KUKA KRL program: MyProgram_070().src

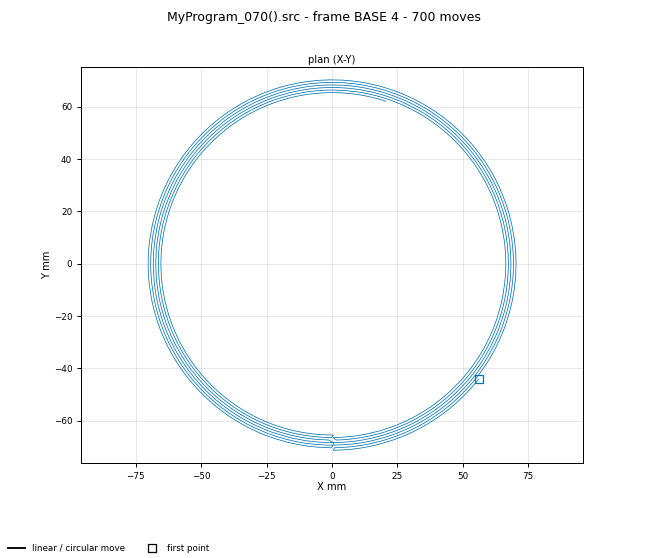
[picture p0: tool path of MyProgram_070().src in frame BASE 4, 700 of 700 moves have a stored position in this frame; points joined in program order, loops and branches not executed]
&ACCESS RVP
&REL 1
&PARAM TEMPLATE = C:\KRC\Roboter\Template\vorgabe
&PARAM EDITMASK = *
DEF MyProgram_070()
; ---- Setting reference (Base) ----
$BASE = BASE_DATA[4]

; --------------------------
; ---- Setting tool (TCP) ----
$TOOL = TOOL_DATA[3]
; --------------------------

$VEL.CP = VEL_APROX_PRINT
Startdeposition()
$VEL.CP = VEL_PRINT
LIN {X 56.046,Y -44.0463,Z 76,A -44.288,B 24.9035,C -2.2676,E1 25.1245,E2 128.6821} C_DIS
LIN {X 53.7927,Y -46.7714,Z 76,A -47.1061,B 24.9041,C -2.261,E1 25.1194,E2 131.503} C_DIS
LIN {X 51.1521,Y -49.6455,Z 76,A -50.0021,B 24.9041,C -2.2599,E1 25.1139,E2 134.3889} C_DIS
LIN {X 49.3417,Y -51.445,Z 76,A -52.3384,B 24.9053,C -2.2472,E1 25.1092,E2 136.7455} C_DIS
LIN {X 46.445,Y -54.0753,Z 76,A -55.3463,B 24.9056,C -2.2438,E1 25.1029,E2 139.7495} C_DIS
LIN {X 43.668,Y -56.3411,Z 76,A -58.1698,B 24.9059,C -2.2391,E1 25.0967,E2 142.5734} C_DIS
LIN {X 40.701,Y -58.5203,Z 76,A -60.9127,B 24.9059,C -2.239,E1 25.0905,E2 145.307} C_DIS
LIN {X 38.2526,Y -60.15,Z 76,A -63.889,B 24.9077,C -2.2179,E1 25.0835,E2 148.3235} C_DIS
LIN {X 34.8025,Y -62.2092,Z 76,A -67.0175,B 24.908,C -2.2149,E1 25.0759,E2 151.4498} C_DIS
LIN {X 30.8316,Y -64.2698,Z 76,A -70.4455,B 24.908,C -2.2135,E1 25.0673,E2 154.8717} C_DIS
LIN {X 27.6575,Y -65.6982,Z 76,A -73.0295,B 24.908,C -2.2151,E1 25.0607,E2 157.4458} C_DIS
LIN {X 23.6668,Y -67.239,Z 76,A -76.1249,B 24.9076,C -2.2196,E1 25.0527,E2 160.5239} C_DIS
LIN {X 19.5102,Y -68.5606,Z 76,A -79.8203,B 24.9083,C -2.2105,E1 25.0428,E2 164.2341} C_DIS
LIN {X 15.9897,Y -69.466,Z 76,A -83.1017,B 24.9094,C -2.1982,E1 25.0338,E2 167.5398} C_DIS
LIN {X 11.549,Y -70.341,Z 76,A -86.5042,B 24.9091,C -2.2014,E1 25.0245,E2 170.9309} C_DIS
LIN {X 7.3989,Y -70.8975,Z 76,A -90.297,B 24.9102,C -2.1885,E1 25.0139,E2 174.7517} C_DIS
LIN {X 3.8952,Y -71.176,Z 76,A -93.5754,B 24.9112,C -2.1759,E1 25.0047,E2 178.0587} C_DIS
LIN {X 0.4617,Y -71.2706,Z 76,A -93.732,B 24.9057,C -2.2418,E1 25.0047,E2 178.0587} C_DIS
Enddeposition()
LIN {X 0.4617,Y -71.2706,Z 76,A -93.732,B 24.9057,C -2.2418,E1 25.0047,E2 178.0587} C_DIS
Startdeposition()
$VEL.CP = VEL_PRINT
LIN {X 0.982,Y -70.3014,Z 76,A -93.6346,B 24.905,C -2.2498,E1 25.0051,E2 177.9423} C_DIS
LIN {X 4.084,Y -70.1891,Z 76,A -91.6184,B 24.9061,C -2.2376,E1 25.0106,E2 175.9557} C_DIS
LIN {X 7.1431,Y -69.944,Z 76,A -88.5948,B 24.9048,C -2.2524,E1 25.0191,E2 172.8989} C_DIS
LIN {X 11.0153,Y -69.4399,Z 76,A -85.5875,B 24.905,C -2.25,E1 25.0274,E2 169.8999} C_DIS
LIN {X 14.077,Y -68.8839,Z 76,A -83.2844,B 24.9054,C -2.246,E1 25.0337,E2 167.6089} C_DIS
LIN {X 18.31,Y -67.8815,Z 76,A -79.8324,B 24.9053,C -2.247,E1 25.043,E2 164.1596} C_DIS
LIN {X 22.0646,Y -66.756,Z 76,A -76.4652,B 24.9046,C -2.2553,E1 25.052,E2 160.7789} C_DIS
LIN {X 26.987,Y -64.9227,Z 76,A -72.2326,B 24.9042,C -2.2597,E1 25.0631,E2 156.545} C_DIS
LIN {X 30.316,Y -63.4359,Z 76,A -69.0283,B 24.9033,C -2.2706,E1 25.0712,E2 153.3231} C_DIS
LIN {X 33.2683,Y -61.9384,Z 76,A -66.4121,B 24.9031,C -2.2729,E1 25.0777,E2 150.7087} C_DIS
LIN {X 35.6896,Y -60.5757,Z 76,A -64.0683,B 24.9025,C -2.2791,E1 25.0834,E2 148.3573} C_DIS
LIN {X 39.2963,Y -58.3008,Z 76,A -61.2698,B 24.9036,C -2.2674,E1 25.0899,E2 145.5958} C_DIS
LIN {X 41.6342,Y -56.6548,Z 76,A -58.6689,B 24.9025,C -2.2794,E1 25.0958,E2 142.9754} C_DIS
LIN {X 43.4611,Y -55.2659,Z 76,A -56.6561,B 24.9018,C -2.2873,E1 25.1003,E2 140.9513} C_DIS
LIN {X 45.7398,Y -53.3953,Z 76,A -54.201,B 24.9013,C -2.2941,E1 25.1056,E2 138.4896} C_DIS
LIN {X 48.1424,Y -51.2392,Z 76,A -51.4487,B 24.9004,C -2.3035,E1 25.1112,E2 135.7262} C_DIS
LIN {X 50.9425,Y -48.4564,Z 76,A -48.3885,B 24.9001,C -2.307,E1 25.1172,E2 132.671} C_DIS
LIN {X 53.1048,Y -46.077,Z 76,A -45.8317,B 24.8997,C -2.3118,E1 25.1219,E2 130.1142} C_DIS
LIN {X 54.9628,Y -43.8435,Z 76,A -43.5864,B 24.8995,C -2.3146,E1 25.1259,E2 127.8727} C_DIS
LIN {X 56.3842,Y -42.0007,Z 76,A -41.0111,B 24.8974,C -2.3387,E1 25.1303,E2 125.2527} C_DIS
LIN {X 59.0022,Y -38.236,Z 76,A -37.8592,B 24.8979,C -2.3325,E1 25.1351,E2 122.131} C_DIS
LIN {X 60.4071,Y -35.9749,Z 76,A -35.0121,B 24.8957,C -2.3578,E1 25.1393,E2 119.2387} C_DIS
LIN {X 62.0404,Y -33.0792,Z 76,A -33.1188,B 24.897,C -2.3425,E1 25.1417,E2 117.3914} C_DIS
LIN {X 64.037,Y -29.0242,Z 76,A -29.3448,B 24.8958,C -2.356,E1 25.1463,E2 113.606} C_DIS
LIN {X 65.9881,Y -24.2643,Z 76,A -25.2544,B 24.895,C -2.3658,E1 25.1505,E2 109.515} C_DIS
LIN {X 67.3327,Y -20.2366,Z 76,A -22.1313,B 24.8949,C -2.3669,E1 25.1532,E2 106.407} C_DIS
LIN {X 68.3707,Y -16.3915,Z 76,A -18.7483,B 24.8936,C -2.3809,E1 25.1557,E2 103.0104} C_DIS
LIN {X 68.9606,Y -13.7027,Z 76,A -16.1394,B 24.8921,C -2.3983,E1 25.1571,E2 100.3756} C_DIS
LIN {X 69.5706,Y -10.1543,Z 76,A -13.1317,B 24.891,C -2.4097,E1 25.1585,E2 97.3586} C_DIS
LIN {X 70.0627,Y -5.869,Z 76,A -10.1362,B 24.8914,C -2.4061,E1 25.1593,E2 94.3893} C_DIS
LIN {X 70.1901,Y -4.0663,Z 76,A -8.1896,B 24.8897,C -2.4243,E1 25.1596,E2 92.4114} C_DIS
LIN {X 70.307,Y 0.373,Z 76,A -4.9729,B 24.8897,C -2.4243,E1 25.1598,E2 89.2137} C_DIS
LIN {X 70.2315,Y 3.2685,Z 76,A -2.5141,B 24.8888,C -2.4346,E1 25.1595,E2 86.7453} C_DIS
LIN {X 70.0316,Y 6.2221,Z 76,A 0.1607,B 24.8874,C -2.4496,E1 25.1589,E2 84.0509} C_DIS
LIN {X 69.6628,Y 9.5074,Z 76,A 2.8886,B 24.8865,C -2.4589,E1 25.1579,E2 81.317} C_DIS
LIN {X 68.6351,Y 15.2465,Z 76,A 7.2916,B 24.8861,C -2.4637,E1 25.1556,E2 76.9286} C_DIS
LIN {X 67.535,Y 19.5537,Z 76,A 10.9636,B 24.8849,C -2.4759,E1 25.153,E2 73.2488} C_DIS
LIN {X 66.3853,Y 23.1552,Z 76,A 13.9692,B 24.8843,C -2.4829,E1 25.1503,E2 70.2436} C_DIS
LIN {X 64.2148,Y 28.6304,Z 76,A 19.6503,B 24.8807,C -2.5213,E1 25.1441,E2 64.5028} C_DIS
LIN {X 62.527,Y 32.1489,Z 76,A 21.686,B 24.8829,C -2.498,E1 25.1417,E2 62.5332} C_DIS
LIN {X 60.6342,Y 35.5901,Z 76,A 25.5848,B 24.8802,C -2.5259,E1 25.1362,E2 58.5887} C_DIS
LIN {X 58.5935,Y 38.8586,Z 76,A 28.5373,B 24.88,C -2.5287,E1 25.1317,E2 55.6444} C_DIS
LIN {X 56.0964,Y 42.3838,Z 76,A 32.3885,B 24.8783,C -2.5464,E1 25.1253,E2 51.7698} C_DIS
LIN {X 54.0444,Y 44.9706,Z 76,A 33.9936,B 24.8805,C -2.5228,E1 25.1226,E2 50.2279} C_DIS
LIN {X 52.7507,Y 46.4822,Z 76,A 36.1228,B 24.8789,C -2.5403,E1 25.1186,E2 48.0669} C_DIS
LIN {X 50.1679,Y 49.258,Z 76,A 39.0626,B 24.8786,C -2.5429,E1 25.1129,E2 45.1337} C_DIS
LIN {X 47.8972,Y 51.4689,Z 76,A 41.7967,B 24.8777,C -2.5522,E1 25.1074,E2 42.3887} C_DIS
LIN {X 45.0927,Y 53.943,Z 76,A 44.958,B 24.8769,C -2.5611,E1 25.1007,E2 39.2187} C_DIS
LIN {X 42.515,Y 55.9979,Z 76,A 47.7041,B 24.8762,C -2.5675,E1 25.0946,E2 36.4677} C_DIS
LIN {X 39.0202,Y 58.4868,Z 76,A 50.8817,B 24.8765,C -2.5647,E1 25.0873,E2 33.3075} C_DIS
LIN {X 36.5864,Y 60.0383,Z 76,A 53.5411,B 24.8754,C -2.5764,E1 25.0809,E2 30.6288} C_DIS
LIN {X 33.0412,Y 62.0603,Z 76,A 56.6166,B 24.8756,C -2.5742,E1 25.0734,E2 27.5673} C_DIS
LIN {X 29.9797,Y 63.5963,Z 76,A 58.9584,B 24.8764,C -2.5659,E1 25.0676,E2 25.2516} C_DIS
LIN {X 26.8045,Y 64.9983,Z 76,A 61.9409,B 24.8757,C -2.5729,E1 25.06,E2 22.2596} C_DIS
LIN {X 23.6744,Y 66.2031,Z 76,A 64.8951,B 24.8749,C -2.5811,E1 25.0522,E2 19.2922} C_DIS
LIN {X 18.4504,Y 67.8436,Z 76,A 69.8253,B 24.8734,C -2.5963,E1 25.0389,E2 14.3344} C_DIS
LIN {X 14.1564,Y 68.8676,Z 76,A 72.7198,B 24.875,C -2.5802,E1 25.0312,E2 11.4821} C_DIS
LIN {X 10.548,Y 69.5121,Z 76,A 75.8816,B 24.8745,C -2.5856,E1 25.0224,E2 8.3107} C_DIS
LIN {X 7.4548,Y 69.9114,Z 76,A 78.622,B 24.874,C -2.591,E1 25.0148,E2 5.5595} C_DIS
LIN {X 4.0327,Y 70.192,Z 76,A 81.0822,B 24.8748,C -2.5827,E1 25.008,E2 3.1202} C_DIS
LIN {X -0.879,Y 70.3033,Z 76,A 85.4871,B 24.8739,C -2.5919,E1 24.9957,E2 -1.3062} C_DIS
LIN {X -5.2334,Y 70.1135,Z 76,A 89.3521,B 24.8733,C -2.5982,E1 24.9848,E2 -5.1875} C_DIS
LIN {X -9.7766,Y 69.6246,Z 76,A 92.491,B 24.8749,C -2.5818,E1 24.9762,E2 -8.2896} C_DIS
LIN {X -12.8317,Y 69.1278,Z 76,A 95.0643,B 24.8749,C -2.5811,E1 24.9692,E2 -10.8639} C_DIS
LIN {X -17.1436,Y 68.1863,Z 76,A 98.3624,B 24.8759,C -2.5708,E1 24.9602,E2 -14.1416} C_DIS
LIN {X -19.7217,Y 67.4855,Z 76,A 100.7953,B 24.8756,C -2.5746,E1 24.9537,E2 -16.5873} C_DIS
LIN {X -21.8021,Y 66.842,Z 76,A 103.6721,B 24.8732,C -2.5988,E1 24.9459,E2 -19.5271} C_DIS
LIN {X -25.8804,Y 65.3712,Z 76,A 106.5746,B 24.8751,C -2.579,E1 24.9384,E2 -22.3888} C_DIS
LIN {X -30.1889,Y 63.497,Z 76,A 109.6094,B 24.8775,C -2.5548,E1 24.9308,E2 -25.3734} C_DIS
LIN {X -32.3827,Y 62.4061,Z 76,A 111.9885,B 24.8769,C -2.5605,E1 24.9249,E2 -27.7723} C_DIS
LIN {X -35.1346,Y 60.8993,Z 76,A 114.6376,B 24.8771,C -2.5582,E1 24.9184,E2 -30.4236} C_DIS
LIN {X -38.0039,Y 59.1511,Z 76,A 117.0205,B 24.8784,C -2.545,E1 24.9128,E2 -32.7826} C_DIS
LIN {X -40.7946,Y 57.2622,Z 76,A 120.2449,B 24.8779,C -2.5505,E1 24.9054,E2 -36.0311} C_DIS
LIN {X -43.6506,Y 55.1161,Z 76,A 123.2664,B 24.8782,C -2.5469,E1 24.8987,E2 -39.0551} C_DIS
LIN {X -46.6368,Y 52.6145,Z 76,A 126.1926,B 24.8794,C -2.5342,E1 24.8925,E2 -41.9624} C_DIS
LIN {X -49.2236,Y 50.2022,Z 76,A 129.1034,B 24.88,C -2.5282,E1 24.8867,E2 -44.8708} C_DIS
LIN {X -51.5293,Y 47.8313,Z 76,A 132.0741,B 24.88,C -2.5278,E1 24.8809,E2 -47.8535} C_DIS
LIN {X -54.1014,Y 44.9021,Z 76,A 134.7336,B 24.8819,C -2.5082,E1 24.8762,E2 -50.4784} C_DIS
LIN {X -57.0976,Y 41.0253,Z 76,A 138.6959,B 24.883,C -2.497,E1 24.8695,E2 -54.4328} C_DIS
LIN {X -59.4927,Y 37.4669,Z 76,A 142.5436,B 24.8831,C -2.4951,E1 24.8635,E2 -58.2952} C_DIS
LIN {X -62.3377,Y 32.5154,Z 76,A 147.0699,B 24.8847,C -2.4789,E1 24.8574,E2 -62.8066} C_DIS
LIN {X -64.3342,Y 28.3611,Z 76,A 151.3266,B 24.8847,C -2.4788,E1 24.8523,E2 -67.0861} C_DIS
LIN {X -65.9894,Y 24.2609,Z 76,A 155.085,B 24.8854,C -2.4712,E1 24.8486,E2 -70.8478} C_DIS
LIN {X -67.3651,Y 20.1274,Z 76,A 158.0786,B 24.8875,C -2.4482,E1 24.8461,E2 -73.8034} C_DIS
LIN {X -68.6256,Y 15.2897,Z 76,A 162.3819,B 24.8882,C -2.4404,E1 24.8432,E2 -78.1132} C_DIS
LIN {X -69.7157,Y 9.1042,Z 76,A 167.4567,B 24.8898,C -2.4232,E1 24.8409,E2 -83.1772} C_DIS
LIN {X -70.047,Y 6.0611,Z 76,A 170.0826,B 24.8903,C -2.4181,E1 24.8402,E2 -85.8067} C_DIS
LIN {X -70.2593,Y 2.6331,Z 76,A 173.3158,B 24.8903,C -2.4187,E1 24.8398,E2 -89.0608} C_DIS
LIN {X -70.289,Y -1.6562,Z 76,A 176.3465,B 24.8921,C -2.3975,E1 24.8398,E2 -92.059} C_DIS
LIN {X -70.1616,Y -4.5333,Z 76,A 178.3177,B 24.8935,C -2.382,E1 24.8402,E2 -94.005} C_DIS
LIN {X -69.8624,Y -7.9038,Z 76,A -178.0713,B 24.8926,C -2.392,E1 24.8412,E2 -97.6615} C_DIS
LIN {X -69.026,Y -13.3629,Z 76,A -174.6364,B 24.896,C -2.3548,E1 24.8427,E2 -101.0279} C_DIS
LIN {X -68.3416,Y -16.5107,Z 76,A -171.6433,B 24.896,C -2.3548,E1 24.8445,E2 -104.0386} C_DIS
LIN {X -67.9223,Y -18.159,Z 76,A -169.0025,B 24.8939,C -2.3783,E1 24.8465,E2 -106.751} C_DIS
LIN {X -66.7452,Y -22.0992,Z 76,A -166.6384,B 24.8967,C -2.3465,E1 24.8485,E2 -109.0526} C_DIS
LIN {X -65.5626,Y -25.3915,Z 76,A -163.6616,B 24.8972,C -2.341,E1 24.8514,E2 -112.0331} C_DIS
LIN {X -63.7317,Y -29.6889,Z 76,A -160.4081,B 24.8992,C -2.3181,E1 24.855,E2 -115.2498} C_DIS
LIN {X -62.8366,Y -31.5412,Z 76,A -157.8748,B 24.8979,C -2.3325,E1 24.8582,E2 -117.8311} C_DIS
LIN {X -60.4425,Y -35.9149,Z 76,A -154.2301,B 24.8997,C -2.3123,E1 24.8632,E2 -121.4469} C_DIS
LIN {X -58.459,Y -39.0595,Z 76,A -151.0903,B 24.9001,C -2.3071,E1 24.8679,E2 -124.5899} C_DIS
LIN {X -56.3005,Y -42.1121,Z 76,A -148.2796,B 24.9012,C -2.2943,E1 24.8725,E2 -127.3839} C_DIS
LIN {X -53.8835,Y -45.1642,Z 76,A -144.8399,B 24.9014,C -2.2929,E1 24.8785,E2 -130.8364} C_DIS
LIN {X -50.8955,Y -48.5073,Z 76,A -140.7895,B 24.9013,C -2.2941,E1 24.8862,E2 -134.9073} C_DIS
LIN {X -47.7104,Y -51.6423,Z 76,A -136.9969,B 24.9016,C -2.2902,E1 24.8939,E2 -138.7063} C_DIS
LIN {X -44.4592,Y -54.4665,Z 76,A -133.5833,B 24.9024,C -2.2814,E1 24.9012,E2 -142.1121} C_DIS
LIN {X -40.1072,Y -57.7457,Z 76,A -129.7925,B 24.9043,C -2.2586,E1 24.9097,E2 -145.862} C_DIS
LIN {X -38.5819,Y -58.776,Z 76,A -127.6352,B 24.9032,C -2.2718,E1 24.9148,E2 -148.0577} C_DIS
LIN {X -34.29,Y -61.3787,Z 76,A -123.8725,B 24.9043,C -2.2582,E1 24.9238,E2 -151.7994} C_DIS
LIN {X -32.1773,Y -62.5125,Z 76,A -121.4445,B 24.9036,C -2.2672,E1 24.9299,E2 -154.2552} C_DIS
LIN {X -28.0715,Y -64.4604,Z 76,A -118.1956,B 24.9049,C -2.2521,E1 24.9381,E2 -157.4762} C_DIS
LIN {X -25.0883,Y -65.6793,Z 76,A -115.3143,B 24.9045,C -2.2558,E1 24.9456,E2 -160.3725} C_DIS
LIN {X -21.3698,Y -66.9819,Z 76,A -111.9034,B 24.9043,C -2.2582,E1 24.9547,E2 -163.7954} C_DIS
LIN {X -17.1875,Y -68.1751,Z 76,A -108.9664,B 24.9058,C -2.2411,E1 24.9625,E2 -166.6962} C_DIS
LIN {X -13.1189,Y -69.073,Z 76,A -105.0438,B 24.9048,C -2.2527,E1 24.9733,E2 -170.6511} C_DIS
LIN {X -8.7588,Y -69.7604,Z 76,A -101.7384,B 24.9055,C -2.2446,E1 24.9824,E2 -173.9399} C_DIS
LIN {X -5.1259,Y -70.1203,Z 76,A -98.2447,B 24.9044,C -2.2577,E1 24.9922,E2 -177.4662} C_DIS
LIN {X -0.3551,Y -70.3067,Z 76,A -95.0784,B 24.9059,C -2.2398,E1 25.001,E2 -180.5903} C_DIS
LIN {X -0.3551,Y -70.3067,Z 76,A -95.0784,B 24.9059,C -2.2398,E1 25.001,E2 -180.5903} C_DIS
Enddeposition()
LIN {X 0.4577,Y -69.3289,Z 76,A -95.2886,B 24.9063,C -2.235,E1 25.0003,E2 -180.3688} C_DIS
Startdeposition()
$VEL.CP = VEL_PRINT
LIN {X -2.2981,Y -69.2948,Z 76,A -98.0999,B 24.9074,C -2.2216,E1 24.9924,E2 -177.5252} C_DIS
LIN {X -6.6522,Y -69.0134,Z 76,A -101.4214,B 24.9068,C -2.2285,E1 24.9832,E2 -174.2188} C_DIS
LIN {X -10.3753,Y -68.5523,Z 76,A -104.6477,B 24.907,C -2.2261,E1 24.9742,E2 -170.9843} C_DIS
LIN {X -14.0152,Y -67.9014,Z 76,A -107.745,B 24.907,C -2.2263,E1 24.9657,E2 -167.884} C_DIS
LIN {X -17.4504,Y -67.101,Z 76,A -110.7104,B 24.907,C -2.2267,E1 24.9577,E2 -164.9153} C_DIS
LIN {X -20.8924,Y -66.111,Z 76,A -113.5911,B 24.9067,C -2.2306,E1 24.95,E2 -162.0391} C_DIS
LIN {X -24.9256,Y -64.6984,Z 76,A -117.4459,B 24.907,C -2.2262,E1 24.9399,E2 -158.166} C_DIS
LIN {X -29.0062,Y -62.9741,Z 76,A -120.9638,B 24.9064,C -2.2334,E1 24.9309,E2 -154.6568} C_DIS
LIN {X -32.2075,Y -61.3979,Z 76,A -123.8427,B 24.906,C -2.2387,E1 24.9238,E2 -151.7828} C_DIS
LIN {X -36.2337,Y -59.1118,Z 76,A -127.9093,B 24.906,C -2.2387,E1 24.914,E2 -147.7038} C_DIS
LIN {X -39.375,Y -57.0674,Z 76,A -131.2209,B 24.906,C -2.2388,E1 24.9063,E2 -144.3814} C_DIS
LIN {X -41.9767,Y -55.1828,Z 76,A -133.8285,B 24.9055,C -2.2445,E1 24.9005,E2 -141.7778} C_DIS
LIN {X -44.7872,Y -52.9261,Z 76,A -136.5323,B 24.9045,C -2.2561,E1 24.8947,E2 -139.0914} C_DIS
LIN {X -47.9128,Y -50.1145,Z 76,A -140.2271,B 24.9043,C -2.2582,E1 24.8872,E2 -135.3865} C_DIS
LIN {X -50.247,Y -47.7745,Z 76,A -143.3604,B 24.9046,C -2.2553,E1 24.8811,E2 -132.2327} C_DIS
LIN {X -52.7672,Y -44.9738,Z 76,A -145.3265,B 24.9019,C -2.2872,E1 24.8776,E2 -130.334} C_DIS
LIN {X -55.0871,Y -42.1012,Z 76,A -148.3985,B 24.9013,C -2.2939,E1 24.8723,E2 -127.2634} C_DIS
LIN {X -57.0012,Y -39.4702,Z 76,A -151.8103,B 24.9021,C -2.2849,E1 24.8667,E2 -123.8133} C_DIS
LIN {X -59.2985,Y -35.9265,Z 76,A -155.0154,B 24.9008,C -2.2999,E1 24.862,E2 -120.628} C_DIS
LIN {X -61.0832,Y -32.8017,Z 76,A -157.9285,B 24.9,C -2.3092,E1 24.858,E2 -117.7215} C_DIS
LIN {X -62.7153,Y -29.5621,Z 76,A -160.5487,B 24.8985,C -2.3255,E1 24.8548,E2 -115.1261} C_DIS
LIN {X -63.9481,Y -26.7896,Z 76,A -164.0441,B 24.8997,C -2.3116,E1 24.8509,E2 -111.5783} C_DIS
LIN {X -65.4565,Y -22.8577,Z 76,A -166.9216,B 24.8978,C -2.3344,E1 24.8482,E2 -108.739} C_DIS
LIN {X -66.5411,Y -19.4743,Z 76,A -169.8141,B 24.8969,C -2.344,E1 24.8458,E2 -105.8528} C_DIS
LIN {X -67.3942,Y -16.2808,Z 76,A -172.9161,B 24.8969,C -2.3445,E1 24.8437,E2 -102.7338} C_DIS
LIN {X -68.0566,Y -13.2416,Z 76,A -175.3894,B 24.896,C -2.3544,E1 24.8423,E2 -100.2695} C_DIS
LIN {X -68.898,Y -7.7571,Z 76,A -179.8118,B 24.8944,C -2.372,E1 24.8406,E2 -95.8629} C_DIS
LIN {X -69.2396,Y -3.5982,Z 76,A 176.8648,B 24.8932,C -2.3855,E1 24.8399,E2 -92.5517} C_DIS
LIN {X -69.3292,Y -0.7837,Z 76,A 174.0646,B 24.8934,C -2.383,E1 24.8398,E2 -89.7286} C_DIS
LIN {X -69.2747,Y 2.8367,Z 76,A 171.1734,B 24.8924,C -2.3946,E1 24.84,E2 -86.8477} C_DIS
LIN {X -68.9605,Y 7.174,Z 76,A 167.9411,B 24.8907,C -2.4135,E1 24.8408,E2 -83.6412} C_DIS
LIN {X -68.4487,Y 11.0432,Z 76,A 163.9597,B 24.8912,C -2.408,E1 24.8424,E2 -79.623} C_DIS
LIN {X -67.8399,Y 14.3125,Z 76,A 161.4759,B 24.8899,C -2.4221,E1 24.8438,E2 -77.1582} C_DIS
LIN {X -66.8926,Y 18.2303,Z 76,A 158.2227,B 24.8888,C -2.4341,E1 24.846,E2 -73.9147} C_DIS
LIN {X -65.032,Y 24.0406,Z 76,A 153.315,B 24.8871,C -2.4524,E1 24.8503,E2 -69.0226} C_DIS
LIN {X -63.367,Y 28.1386,Z 76,A 149.0704,B 24.8872,C -2.451,E1 24.855,E2 -64.7513} C_DIS
LIN {X -61.336,Y 32.3251,Z 76,A 145.3728,B 24.8859,C -2.4653,E1 24.8596,E2 -61.0681} C_DIS
LIN {X -59.9501,Y 34.8298,Z 76,A 143.3098,B 24.8847,C -2.4784,E1 24.8625,E2 -59.0255} C_DIS
LIN {X -57.8712,Y 38.1829,Z 76,A 139.7973,B 24.8844,C -2.4822,E1 24.8678,E2 -55.5042} C_DIS
LIN {X -55.9088,Y 41.0026,Z 76,A 136.3212,B 24.8849,C -2.4764,E1 24.8735,E2 -51.9975} C_DIS
LIN {X -53.5749,Y 44.0103,Z 76,A 134.3281,B 24.8818,C -2.5089,E1 24.8769,E2 -50.0727} C_DIS
LIN {X -51.1558,Y 46.7983,Z 76,A 130.788,B 24.8821,C -2.5061,E1 24.8835,E2 -46.51} C_DIS
LIN {X -48.3201,Y 49.7204,Z 76,A 127.2624,B 24.8817,C -2.5107,E1 24.8904,E2 -42.9803} C_DIS
LIN {X -45.522,Y 52.2951,Z 76,A 124.031,B 24.8812,C -2.5158,E1 24.8972,E2 -39.7484} C_DIS
LIN {X -41.9323,Y 55.2162,Z 76,A 120.7541,B 24.8793,C -2.5358,E1 24.9043,E2 -36.507} C_DIS
LIN {X -40.2407,Y 56.4597,Z 76,A 118.5877,B 24.8799,C -2.5299,E1 24.9092,E2 -34.3189} C_DIS
LIN {X -37.3743,Y 58.3968,Z 76,A 115.5171,B 24.8798,C -2.5306,E1 24.9165,E2 -31.2402} C_DIS
LIN {X -33.2117,Y 60.8607,Z 76,A 112.0893,B 24.8779,C -2.5502,E1 24.9247,E2 -27.8488} C_DIS
LIN {X -30.6958,Y 62.1675,Z 76,A 109.8559,B 24.8773,C -2.5564,E1 24.9302,E2 -25.6243} C_DIS
LIN {X -27.4552,Y 63.6655,Z 76,A 106.4729,B 24.8778,C -2.5511,E1 24.9389,E2 -22.2202} C_DIS
LIN {X -23.8022,Y 65.1189,Z 76,A 103.044,B 24.8778,C -2.5513,E1 24.9478,E2 -18.7847} C_DIS
LIN {X -20.9233,Y 66.1014,Z 76,A 100.8133,B 24.8769,C -2.5606,E1 24.9537,E2 -16.5721} C_DIS
LIN {X -16.4685,Y 67.3484,Z 76,A 97.2474,B 24.876,C -2.5704,E1 24.9633,E2 -13.024} C_DIS
LIN {X -14.5908,Y 67.7802,Z 76,A 95.2499,B 24.8767,C -2.5624,E1 24.9688,E2 -11.0051} C_DIS
LIN {X -10.6098,Y 68.516,Z 76,A 92.2784,B 24.8757,C -2.5735,E1 24.9769,E2 -8.0572} C_DIS
LIN {X -8.4286,Y 68.8194,Z 76,A 89.984,B 24.8766,C -2.5635,E1 24.9833,E2 -5.7374} C_DIS
LIN {X -5.0436,Y 69.1499,Z 76,A 87.6995,B 24.8753,C -2.5772,E1 24.9896,E2 -3.4842} C_DIS
LIN {X -0.7036,Y 69.3296,Z 76,A 84.2345,B 24.8749,C -2.5813,E1 24.9992,E2 -0.0282} C_DIS
LIN {X 4.2736,Y 69.202,Z 76,A 79.1496,B 24.8771,C -2.5584,E1 25.0136,E2 5.1096} C_DIS
LIN {X 9.2555,Y 68.713,Z 76,A 75.3268,B 24.8765,C -2.5652,E1 25.0241,E2 8.9135} C_DIS
LIN {X 12.8495,Y 68.1321,Z 76,A 72.6393,B 24.8758,C -2.572,E1 25.0314,E2 11.5821} C_DIS
LIN {X 16.4871,Y 67.3433,Z 76,A 69.5818,B 24.8759,C -2.5709,E1 25.0398,E2 14.638} C_DIS
LIN {X 19.7414,Y 66.4627,Z 76,A 66.3796,B 24.8771,C -2.5587,E1 25.0484,E2 17.8637} C_DIS
LIN {X 24.3673,Y 64.9099,Z 76,A 62.5542,B 24.8769,C -2.5603,E1 25.0585,E2 21.6775} C_DIS
LIN {X 28.4211,Y 63.2397,Z 76,A 59.2303,B 24.8766,C -2.564,E1 25.067,E2 24.9847} C_DIS
LIN {X 31.1865,Y 61.9238,Z 76,A 56.1416,B 24.8782,C -2.5469,E1 25.0748,E2 28.1059} C_DIS
LIN {X 35.9498,Y 59.2844,Z 76,A 52.3995,B 24.877,C -2.5599,E1 25.0838,E2 31.806} C_DIS
LIN {X 38.547,Y 57.6299,Z 76,A 49.4918,B 24.8783,C -2.5466,E1 25.0906,E2 34.7356} C_DIS
LIN {X 41.5541,Y 55.5003,Z 76,A 46.6437,B 24.8783,C -2.5466,E1 25.097,E2 37.5739} C_DIS
LIN {X 44.8521,Y 52.8708,Z 76,A 42.7236,B 24.88,C -2.5288,E1 25.1056,E2 41.521} C_DIS
LIN {X 47.6599,Y 50.3548,Z 76,A 40.1893,B 24.8791,C -2.5377,E1 25.1107,E2 44.0239} C_DIS
LIN {X 50.0162,Y 48.0147,Z 76,A 36.8652,B 24.8811,C -2.5167,E1 25.1173,E2 47.3835} C_DIS
LIN {X 52.8409,Y 44.8872,Z 76,A 34.0411,B 24.8802,C -2.5263,E1 25.1225,E2 50.1724} C_DIS
LIN {X 55.0308,Y 42.1742,Z 76,A 30.7178,B 24.882,C -2.5078,E1 25.1283,E2 53.5239} C_DIS
LIN {X 57.4534,Y 38.8089,Z 76,A 27.7605,B 24.8816,C -2.5118,E1 25.133,E2 56.4572} C_DIS
LIN {X 58.5809,Y 37.0856,Z 76,A 25.4838,B 24.8834,C -2.4921,E1 25.1365,E2 58.7691} C_DIS
LIN {X 61.0086,Y 32.9391,Z 76,A 21.8858,B 24.8834,C -2.4915,E1 25.1414,E2 62.3497} C_DIS
LIN {X 62.5805,Y 29.8444,Z 76,A 19.0341,B 24.8842,C -2.4841,E1 25.1449,E2 65.2038} C_DIS
LIN {X 63.8075,Y 27.1232,Z 76,A 16.4365,B 24.8852,C -2.4736,E1 25.1479,E2 67.812} C_DIS
LIN {X 65.1045,Y 23.8417,Z 76,A 13.1889,B 24.8868,C -2.4562,E1 25.1511,E2 71.0826} C_DIS
LIN {X 66.5647,Y 19.3977,Z 76,A 9.8108,B 24.8866,C -2.458,E1 25.1539,E2 74.4374} C_DIS
LIN {X 67.4168,Y 16.1881,Z 76,A 7.2708,B 24.8869,C -2.4553,E1 25.1556,E2 76.9691} C_DIS
LIN {X 68.1809,Y 12.5893,Z 76,A 4.024,B 24.8882,C -2.4403,E1 25.1574,E2 80.2323} C_DIS
LIN {X 68.707,Y 9.3014,Z 76,A 1.5994,B 24.8882,C -2.4407,E1 25.1585,E2 82.6417} C_DIS
LIN {X 69.1876,Y 4.4869,Z 76,A -3.0622,B 24.891,C -2.41,E1 25.1596,E2 87.3481} C_DIS
LIN {X 69.3188,Y 1.3883,Z 76,A -5.1647,B 24.8906,C -2.4145,E1 25.1598,E2 89.4276} C_DIS
LIN {X 69.2706,Y -2.9325,Z 76,A -8.1908,B 24.8903,C -2.4182,E1 25.1596,E2 92.427} C_DIS
LIN {X 69.0671,Y -6.0699,Z 76,A -11.3953,B 24.8925,C -2.3932,E1 25.159,E2 95.6715} C_DIS
LIN {X 68.6845,Y -9.4594,Z 76,A -14.0422,B 24.8929,C -2.389,E1 25.1581,E2 98.3128} C_DIS
LIN {X 68.2719,Y -12.0832,Z 76,A -16.8467,B 24.895,C -2.3653,E1 25.1567,E2 101.1566} C_DIS
LIN {X 67.6402,Y -15.2303,Z 76,A -20.0415,B 24.8971,C -2.3422,E1 25.1548,E2 104.3875} C_DIS
LIN {X 66.5522,Y -19.4397,Z 76,A -22.1428,B 24.8944,C -2.3717,E1 25.1532,E2 106.407} C_DIS
LIN {X 65.2999,Y -23.304,Z 76,A -25.5652,B 24.8955,C -2.3596,E1 25.1502,E2 109.8387} C_DIS
LIN {X 64.5193,Y -25.3826,Z 76,A -27.471,B 24.8962,C -2.352,E1 25.1483,E2 111.7518} C_DIS
LIN {X 63.5066,Y -27.8199,Z 76,A -30.6116,B 24.8991,C -2.3194,E1 25.1448,E2 114.9524} C_DIS
LIN {X 61.9999,Y -31.0339,Z 76,A -32.6789,B 24.8978,C -2.3342,E1 25.1423,E2 116.9735} C_DIS
LIN {X 59.3611,Y -35.8235,Z 76,A -37.1293,B 24.8987,C -2.3231,E1 25.1362,E2 121.4271} C_DIS
LIN {X 57.8561,Y -38.2059,Z 76,A -39.736,B 24.9,C -2.3091,E1 25.1322,E2 124.0539} C_DIS
LIN {X 55.6973,Y -41.2916,Z 76,A -42.6506,B 24.9002,C -2.306,E1 25.1275,E2 126.9616} C_DIS
LIN {X 53.8756,Y -43.6399,Z 76,A -44.9104,B 24.9003,C -2.3049,E1 25.1236,E2 129.2135} C_DIS
LIN {X 52.4168,Y -45.3827,Z 76,A -46.8787,B 24.901,C -2.2976,E1 25.12,E2 131.19} C_DIS
LIN {X 50.7314,Y -47.2586,Z 76,A -48.9592,B 24.9014,C -2.2925,E1 25.1161,E2 133.2734} C_DIS
LIN {X 48.8647,Y -49.1864,Z 76,A -51.1456,B 24.9018,C -2.288,E1 25.1118,E2 135.4611} C_DIS
LIN {X 46.9337,Y -51.0319,Z 76,A -53.2933,B 24.9021,C -2.2844,E1 25.1074,E2 137.6084} C_DIS
LIN {X 45.0346,Y -52.7153,Z 76,A -55.3629,B 24.9024,C -2.2804,E1 25.103,E2 139.6794} C_DIS
LIN {X 43.2534,Y -54.1865,Z 76,A -57.3741,B 24.903,C -2.2736,E1 25.0987,E2 141.6992} C_DIS
LIN {X 40.9127,Y -55.9747,Z 76,A -59.9704,B 24.9038,C -2.2642,E1 25.0928,E2 144.3083} C_DIS
LIN {X 37.8696,Y -58.0778,Z 76,A -62.8938,B 24.904,C -2.2617,E1 25.0861,E2 147.2278} C_DIS
LIN {X 35.467,Y -59.5748,Z 76,A -64.7926,B 24.9034,C -2.269,E1 25.0816,E2 149.1034} C_DIS
LIN {X 31.5647,Y -61.7308,Z 76,A -68.8805,B 24.9049,C -2.2521,E1 25.0715,E2 153.2195} C_DIS
LIN {X 28.4999,Y -63.2042,Z 76,A -71.5245,B 24.9049,C -2.2521,E1 25.0648,E2 155.8569} C_DIS
LIN {X 25.0079,Y -64.6655,Z 76,A -74.9735,B 24.9059,C -2.2394,E1 25.0558,E2 159.328} C_DIS
LIN {X 21.1283,Y -66.0353,Z 76,A -78.4755,B 24.9065,C -2.2326,E1 25.0466,E2 162.8392} C_DIS
LIN {X 18.2829,Y -66.879,Z 76,A -81.5186,B 24.908,C -2.2151,E1 25.0383,E2 165.9189} C_DIS
LIN {X 14.6185,Y -67.7742,Z 76,A -83.4064,B 24.9056,C -2.2432,E1 25.0333,E2 167.7376} C_DIS
LIN {X 11.2368,Y -68.4163,Z 76,A -86.5176,B 24.9064,C -2.2341,E1 25.0247,E2 170.8667} C_DIS
LIN {X 8.6383,Y -68.7925,Z 76,A -88.8291,B 24.9068,C -2.2292,E1 25.0183,E2 173.188} C_DIS
LIN {X 5.1544,Y -69.1417,Z 76,A -92.1476,B 24.9078,C -2.2172,E1 25.009,E2 176.5331} C_DIS
LIN {X 0.8279,Y -69.3289,Z 76,A -95.2702,B 24.9069,C -2.2273,E1 25.0003,E2 179.6312} C_DIS
LIN {X 0.8279,Y -69.3289,Z 76,A -95.2702,B 24.9069,C -2.2273,E1 25.0003,E2 179.6312} C_DIS
Enddeposition()
LIN {X 0.4414,Y -68.3554,Z 76,A -94.4227,B 24.9031,C -2.273,E1 25.003,E2 178.6753} C_DIS
Startdeposition()
$VEL.CP = VEL_PRINT
LIN {X 3.0198,Y -68.291,Z 76,A -91.8935,B 24.9022,C -2.2829,E1 25.0101,E2 176.1233} C_DIS
LIN {X 6.6757,Y -68.0319,Z 76,A -89.2202,B 24.903,C -2.2744,E1 25.0175,E2 173.4716} C_DIS
LIN {X 9.69,Y -67.6675,Z 76,A -86.5094,B 24.9025,C -2.2802,E1 25.025,E2 170.7492} C_DIS
LIN {X 12.6278,Y -67.1817,Z 76,A -84.1873,B 24.9027,C -2.2777,E1 25.0314,E2 168.4355} C_DIS
LIN {X 15.3225,Y -66.6183,Z 76,A -81.24,B 24.9011,C -2.2962,E1 25.0395,E2 165.4483} C_DIS
LIN {X 20.1854,Y -65.3095,Z 76,A -77.0727,B 24.9008,C -2.2995,E1 25.0507,E2 161.2804} C_DIS
LIN {X 24.9786,Y -63.6306,Z 76,A -73.0552,B 24.9008,C -2.2989,E1 25.0612,E2 157.2729} C_DIS
LIN {X 28.5301,Y -62.1203,Z 76,A -70.4488,B 24.9018,C -2.2873,E1 25.0678,E2 154.7002} C_DIS
LIN {X 30.3859,Y -61.233,Z 76,A -68.6185,B 24.9014,C -2.2928,E1 25.0724,E2 152.8617} C_DIS
LIN {X 32.4973,Y -60.1391,Z 76,A -65.8518,B 24.8993,C -2.3166,E1 25.0793,E2 150.0467} C_DIS
LIN {X 36.4161,Y -57.8507,Z 76,A -61.9364,B 24.8984,C -2.3266,E1 25.0886,E2 146.1199} C_DIS
LIN {X 39.1665,Y -56.0249,Z 76,A -59.9963,B 24.8999,C -2.31,E1 25.093,E2 144.2256} C_DIS
LIN {X 41.6504,Y -54.2036,Z 76,A -57.2129,B 24.8989,C -2.3208,E1 25.0993,E2 141.4268} C_DIS
LIN {X 44.3295,Y -52.0353,Z 76,A -54.3201,B 24.8984,C -2.3273,E1 25.1055,E2 138.5298} C_DIS
LIN {X 47.0032,Y -49.6341,Z 76,A -51.3969,B 24.898,C -2.3319,E1 25.1115,E2 135.6076} C_DIS
LIN {X 49.3112,Y -47.3413,Z 76,A -48.6244,B 24.8973,C -2.3397,E1 25.1169,E2 132.8284} C_DIS
LIN {X 51.7288,Y -44.6883,Z 76,A -45.6686,B 24.8967,C -2.3458,E1 25.1224,E2 129.8713} C_DIS
LIN {X 53.988,Y -41.9303,Z 76,A -42.6993,B 24.8961,C -2.3532,E1 25.1276,E2 126.8986} C_DIS
LIN {X 56.2259,Y -38.8775,Z 76,A -39.2185,B 24.8946,C -2.3702,E1 25.1332,E2 123.3944} C_DIS
LIN {X 58.3125,Y -35.6716,Z 76,A -35.9436,B 24.8936,C -2.3811,E1 25.1381,E2 120.1103} C_DIS
LIN {X 60.5351,Y -31.7536,Z 76,A -32.9735,B 24.8946,C -2.3699,E1 25.142,E2 117.1823} C_DIS
LIN {X 62.4962,Y -27.698,Z 76,A -28.8864,B 24.8929,C -2.3895,E1 25.1469,E2 113.0708} C_DIS
LIN {X 63.6847,Y -24.8408,Z 76,A -26.3133,B 24.8922,C -2.3968,E1 25.1496,E2 110.4946} C_DIS
LIN {X 65.4925,Y -19.5841,Z 76,A -22.2007,B 24.8922,C -2.3961,E1 25.1532,E2 106.407} C_DIS
LIN {X 66.4044,Y -16.2244,Z 76,A -18.7917,B 24.8902,C -2.4187,E1 25.1557,E2 102.9643} C_DIS
LIN {X 67.0275,Y -13.4227,Z 76,A -16.5713,B 24.89,C -2.4211,E1 25.157,E2 100.751} C_DIS
LIN {X 67.5416,Y -10.5316,Z 76,A -13.8818,B 24.8887,C -2.4353,E1 25.1582,E2 98.044} C_DIS
LIN {X 67.9402,Y -7.5534,Z 76,A -11.5365,B 24.8884,C -2.4384,E1 25.159,E2 95.705} C_DIS
LIN {X 68.2438,Y -3.9455,Z 76,A -8.5919,B 24.8877,C -2.4456,E1 25.1596,E2 92.761} C_DIS
LIN {X 68.3576,Y -0.2807,Z 76,A -5.4394,B 24.8866,C -2.4575,E1 25.1598,E2 89.599} C_DIS
LIN {X 68.3187,Y 2.3214,Z 76,A -3.1092,B 24.8856,C -2.4686,E1 25.1596,E2 87.2566} C_DIS
LIN {X 68.0439,Y 6.5485,Z 76,A 0.2979,B 24.885,C -2.4757,E1 25.1589,E2 83.8527} C_DIS
LIN {X 67.7507,Y 9.0953,Z 76,A 2.7093,B 24.8837,C -2.4897,E1 25.158,E2 81.4226} C_DIS
LIN {X 67.0206,Y 13.4532,Z 76,A 6.1567,B 24.8832,C -2.494,E1 25.1563,E2 77.9851} C_DIS
LIN {X 66.0811,Y 17.4952,Z 76,A 9.6454,B 24.8822,C -2.5048,E1 25.1539,E2 74.4911} C_DIS
LIN {X 65.2731,Y 20.3028,Z 76,A 11.8248,B 24.8822,C -2.5048,E1 25.1522,E2 72.3243} C_DIS
LIN {X 64.1123,Y 23.7167,Z 76,A 14.7091,B 24.8818,C -2.5098,E1 25.1495,E2 69.4442} C_DIS
LIN {X 62.955,Y 26.6357,Z 76,A 17.7688,B 24.8799,C -2.529,E1 25.1463,E2 66.3561} C_DIS
LIN {X 61.0099,Y 30.8329,Z 76,A 21.4404,B 24.8795,C -2.5341,E1 25.1418,E2 62.6922} C_DIS
LIN {X 59.9928,Y 32.7671,Z 76,A 23.6145,B 24.8781,C -2.5483,E1 25.1389,E2 60.4959} C_DIS
LIN {X 57.3162,Y 37.253,Z 76,A 27.568,B 24.8781,C -2.5481,E1 25.1332,E2 56.5628} C_DIS
LIN {X 55.2155,Y 40.2993,Z 76,A 30.909,B 24.8768,C -2.5622,E1 25.1277,E2 53.2048} C_DIS
LIN {X 52.6154,Y 43.6395,Z 76,A 34.0003,B 24.8771,C -2.5584,E1 25.1224,E2 50.137} C_DIS
LIN {X 50.5616,Y 46.0042,Z 76,A 36.6787,B 24.8764,C -2.5657,E1 25.1174,E2 47.4534} C_DIS
LIN {X 47.6632,Y 49.001,Z 76,A 40.2544,B 24.8755,C -2.5752,E1 25.1104,E2 43.8704} C_DIS
LIN {X 45.3333,Y 51.1644,Z 76,A 42.7498,B 24.8755,C -2.576,E1 25.1053,E2 41.3831} C_DIS
LIN {X 41.9501,Y 53.9726,Z 76,A 46.6028,B 24.8743,C -2.5872,E1 25.0969,E2 37.5183} C_DIS
LIN {X 39.3978,Y 55.8635,Z 76,A 50.0925,B 24.8718,C -2.6132,E1 25.0889,E2 33.9791} C_DIS
LIN {X 36.4736,Y 57.8148,Z 76,A 52.2258,B 24.8734,C -2.5967,E1 25.084,E2 31.892} C_DIS
LIN {X 33.0392,Y 59.8439,Z 76,A 55.9107,B 24.8721,C -2.6101,E1 25.075,E2 28.1862} C_DIS
LIN {X 29.2434,Y 61.7881,Z 76,A 59.1782,B 24.8724,C -2.6066,E1 25.0668,E2 24.9356} C_DIS
LIN {X 27.2275,Y 62.7013,Z 76,A 61.1063,B 24.872,C -2.6105,E1 25.0619,E2 23.003} C_DIS
LIN {X 22.3623,Y 64.5971,Z 76,A 65.3746,B 24.872,C -2.6118,E1 25.0508,E2 18.7407} C_DIS
LIN {X 20.1246,Y 65.3284,Z 76,A 67.7927,B 24.8707,C -2.6244,E1 25.0442,E2 16.297} C_DIS
LIN {X 16.3317,Y 66.3782,Z 76,A 71.371,B 24.8698,C -2.6333,E1 25.0345,E2 12.703} C_DIS
LIN {X 12.9923,Y 67.1117,Z 76,A 73.149,B 24.8723,C -2.6077,E1 25.0298,E2 10.9879} C_DIS
LIN {X 9.5373,Y 67.6892,Z 76,A 76.8134,B 24.8705,C -2.6264,E1 25.0196,E2 7.2827} C_DIS
LIN {X 6.1242,Y 68.083,Z 76,A 79.0652,B 24.872,C -2.6115,E1 25.0134,E2 5.0678} C_DIS
LIN {X 3.4683,Y 68.2704,Z 76,A 82.3964,B 24.8693,C -2.6381,E1 25.004,E2 1.6746} C_DIS
LIN {X -0.2302,Y 68.3576,Z 76,A 84.1762,B 24.8725,C -2.6058,E1 24.9992,E2 -0.0282} C_DIS
LIN {X -3.1955,Y 68.2831,Z 76,A 87.1652,B 24.8714,C -2.617,E1 24.9908,E2 -3.0442} C_DIS
LIN {X -7.3692,Y 67.9598,Z 76,A 90.547,B 24.8719,C -2.6123,E1 24.9814,E2 -6.4166} C_DIS
LIN {X -9.9017,Y 67.6372,Z 76,A 93.1479,B 24.8709,C -2.6218,E1 24.9742,E2 -9.0421} C_DIS
LIN {X -14.8174,Y 66.733,Z 76,A 96.7213,B 24.8727,C -2.604,E1 24.9645,E2 -12.5773} C_DIS
LIN {X -18.2752,Y 65.8703,Z 76,A 100.5481,B 24.8711,C -2.6205,E1 24.954,E2 -16.449} C_DIS
LIN {X -21.6495,Y 64.8392,Z 76,A 103.1521,B 24.8722,C -2.6089,E1 24.9472,E2 -19.0302} C_DIS
LIN {X -25.3856,Y 63.4706,Z 76,A 106.2276,B 24.8732,C -2.5986,E1 24.9392,E2 -22.0876} C_DIS
LIN {X -29.4495,Y 61.689,Z 76,A 109.9372,B 24.8738,C -2.5928,E1 24.9298,E2 -25.7926} C_DIS
LIN {X -32.6205,Y 60.0723,Z 76,A 113.8359,B 24.8722,C -2.6085,E1 24.9201,E2 -29.7395} C_DIS
LIN {X -35.7746,Y 58.25,Z 76,A 116.0995,B 24.8745,C -2.5853,E1 24.9148,E2 -31.9547} C_DIS
LIN {X -38.3514,Y 56.5858,Z 76,A 118.4037,B 24.8756,C -2.5745,E1 24.9094,E2 -34.2408} C_DIS
LIN {X -40.8253,Y 54.8285,Z 76,A 121.061,B 24.8758,C -2.5719,E1 24.9034,E2 -36.9011} C_DIS
LIN {X -45.3498,Y 51.1496,Z 76,A 125.7753,B 24.8772,C -2.5574,E1 24.8933,E2 -41.5989} C_DIS
LIN {X -47.4275,Y 49.2282,Z 76,A 128.9104,B 24.8761,C -2.5685,E1 24.8869,E2 -44.7734} C_DIS
LIN {X -50.8994,Y 45.6293,Z 76,A 133.1627,B 24.877,C -2.5596,E1 24.8788,E2 -49.0229} C_DIS
LIN {X -53.1836,Y 42.9453,Z 76,A 136.537,B 24.8769,C -2.561,E1 24.8728,E2 -52.4164} C_DIS
LIN {X -55.4144,Y 40.0268,Z 76,A 138.7448,B 24.8795,C -2.534,E1 24.8693,E2 -54.5704} C_DIS
LIN {X -58.1111,Y 35.9992,Z 76,A 142.8993,B 24.8803,C -2.5248,E1 24.8629,E2 -58.7236} C_DIS
LIN {X -59.6485,Y 33.3892,Z 76,A 145.3699,B 24.8812,C -2.5161,E1 24.8595,E2 -61.1864} C_DIS
LIN {X -61.4712,Y 29.9022,Z 76,A 149.0266,B 24.8814,C -2.5141,E1 24.8549,E2 -64.8579} C_DIS
LIN {X -63.8289,Y 24.4689,Z 76,A 153.3669,B 24.884,C -2.486,E1 24.8502,E2 -69.1552} C_DIS
LIN {X -64.8813,Y 21.5246,Z 76,A 156.4036,B 24.884,C -2.4867,E1 24.8474,E2 -72.2109} C_DIS
LIN {X -65.7675,Y 18.639,Z 76,A 159.3283,B 24.8839,C -2.4872,E1 24.8451,E2 -75.1536} C_DIS
LIN {X -66.9554,Y 13.7752,Z 76,A 163.7037,B 24.8848,C -2.4778,E1 24.8424,E2 -79.5324} C_DIS
LIN {X -67.872,Y 8.1368,Z 76,A 167.811,B 24.8875,C -2.4484,E1 24.8408,E2 -83.5938} C_DIS
LIN {X -68.0989,Y 5.9524,Z 76,A 169.8804,B 24.8875,C -2.4473,E1 24.8402,E2 -85.673} C_DIS
LIN {X -68.2902,Y 3.0403,Z 76,A 172.4466,B 24.8881,C -2.4421,E1 24.8399,E2 -88.2421} C_DIS
LIN {X -68.3472,Y -1.2006,Z 76,A 175.8409,B 24.8894,C -2.4274,E1 24.8399,E2 -91.6219} C_DIS
LIN {X -67.9427,Y -7.5329,Z 76,A -178.458,B 24.8902,C -2.4187,E1 24.8411,E2 -97.3364} C_DIS
LIN {X -67.2587,Y -12.2092,Z 76,A -174.7337,B 24.8918,C -2.4015,E1 24.8427,E2 -101.0416} C_DIS
LIN {X -66.6966,Y -14.9832,Z 76,A -171.7066,B 24.8912,C -2.4082,E1 24.8446,E2 -104.1026} C_DIS
LIN {X -65.2044,Y -20.5246,Z 76,A -167.4805,B 24.8936,C -2.3813,E1 24.8478,E2 -108.289} C_DIS
LIN {X -64.2339,Y -23.3835,Z 76,A -165.19,B 24.8947,C -2.3689,E1 24.8499,E2 -110.5627} C_DIS
LIN {X -62.9966,Y -26.537,Z 76,A -161.975,B 24.8947,C -2.3688,E1 24.8533,E2 -113.7954} C_DIS
LIN {X -61.909,Y -28.9842,Z 76,A -159.5262,B 24.8949,C -2.3669,E1 24.8562,E2 -116.2532} C_DIS
LIN {X -60.0419,Y -32.6764,Z 76,A -155.9111,B 24.8954,C -2.3608,E1 24.8609,E2 -119.8728} C_DIS
LIN {X -57.9231,Y -36.3002,Z 76,A -152.8736,B 24.8972,C -2.3412,E1 24.8653,E2 -122.879} C_DIS
LIN {X -54.8123,Y -40.8467,Z 76,A -148.5822,B 24.8988,C -2.3226,E1 24.8721,E2 -127.1474} C_DIS
LIN {X -52.5091,Y -43.7673,Z 76,A -145.1167,B 24.8988,C -2.3229,E1 24.8782,E2 -130.6298} C_DIS
LIN {X -49.5329,Y -47.1107,Z 76,A -141.5671,B 24.8999,C -2.3102,E1 24.8848,E2 -134.1648} C_DIS
LIN {X -47.122,Y -49.5222,Z 76,A -138.7017,B 24.9004,C -2.3044,E1 24.8905,E2 -137.0285} C_DIS
LIN {X -44.2227,Y -52.1263,Z 76,A -135.3884,B 24.9008,C -2.2991,E1 24.8974,E2 -140.3424} C_DIS
LIN {X -41.746,Y -54.1299,Z 76,A -132.0695,B 24.9,C -2.309,E1 24.9047,E2 -143.6971} C_DIS
LIN {X -38.5442,Y -56.4552,Z 76,A -129.1624,B 24.9012,C -2.2942,E1 24.9113,E2 -146.5789} C_DIS
LIN {X -36.9998,Y -57.4787,Z 76,A -127.3676,B 24.901,C -2.2974,E1 24.9156,E2 -148.3871} C_DIS
LIN {X -33.8386,Y -59.3952,Z 76,A -124.0556,B 24.901,C -2.298,E1 24.9236,E2 -151.7104} C_DIS
LIN {X -29.9479,Y -61.4495,Z 76,A -120.6669,B 24.9019,C -2.2864,E1 24.932,E2 -155.0807} C_DIS
LIN {X -25.3659,Y -63.4784,Z 76,A -116.5015,B 24.9024,C -2.2812,E1 24.9427,E2 -159.2434} C_DIS
LIN {X -23.0186,Y -64.3668,Z 76,A -113.8811,B 24.9015,C -2.2917,E1 24.9496,E2 -161.8938} C_DIS
LIN {X -16.4326,Y -66.3536,Z 76,A -109.0397,B 24.9037,C -2.2658,E1 24.9625,E2 -166.6816} C_DIS
LIN {X -14.9288,Y -66.7072,Z 76,A -106.9622,B 24.9021,C -2.284,E1 24.9683,E2 -168.805} C_DIS
LIN {X -10.164,Y -67.5985,Z 76,A -103.3754,B 24.9032,C -2.2712,E1 24.9781,E2 -172.3649} C_DIS
LIN {X -6.7234,Y -68.0274,Z 76,A -99.346,B 24.9009,C -2.2985,E1 24.9894,E2 -176.4614} C_DIS
LIN {X -2.5802,Y -68.3099,Z 76,A -96.8936,B 24.9031,C -2.2732,E1 24.9961,E2 -178.8545} C_DIS
LIN {X 0.4414,Y -68.3554,Z 76,A -94.4212,B 24.9031,C -2.2723,E1 25.003,E2 -181.3246} C_DIS
Enddeposition()
LIN {X 0.4414,Y -68.3554,Z 76,A -94.4212,B 24.9031,C -2.2723,E1 25.003,E2 -181.3246} C_DIS
Startdeposition()
$VEL.CP = VEL_PRINT
LIN {X -1.2393,Y -67.3714,Z 76,A -97.0458,B 24.9042,C -2.26,E1 24.9956,E2 -178.6707} C_DIS
LIN {X -5.685,Y -67.1433,Z 76,A -100.538,B 24.9036,C -2.2667,E1 24.9859,E2 -175.1935} C_DIS
LIN {X -8.4347,Y -66.8532,Z 76,A -103.1777,B 24.9042,C -2.2603,E1 24.9785,E2 -172.5367} C_DIS
LIN {X -12.2725,Y -66.2555,Z 76,A -106.9926,B 24.9051,C -2.2494,E1 24.9679,E2 -168.6924} C_DIS
LIN {X -15.5547,Y -65.5641,Z 76,A -110.2682,B 24.9058,C -2.2412,E1 24.959,E2 -165.3929} C_DIS
LIN {X -19.1776,Y -64.5961,Z 76,A -112.774,B 24.9043,C -2.2588,E1 24.9524,E2 -162.9248} C_DIS
LIN {X -22.6528,Y -63.462,Z 76,A -115.7086,B 24.9037,C -2.2652,E1 24.9446,E2 -159.9998} C_DIS
LIN {X -25.7182,Y -62.2827,Z 76,A -118.7639,B 24.904,C -2.262,E1 24.9367,E2 -156.9302} C_DIS
LIN {X -28.818,Y -60.9108,Z 76,A -121.251,B 24.903,C -2.2741,E1 24.9304,E2 -154.4656} C_DIS
LIN {X -31.1841,Y -59.7332,Z 76,A -124.1151,B 24.9039,C -2.2632,E1 24.9232,E2 -151.5679} C_DIS
LIN {X -35.4669,Y -57.2941,Z 76,A -127.7223,B 24.9023,C -2.282,E1 24.9146,E2 -147.9945} C_DIS
LIN {X -37.8212,Y -55.7674,Z 76,A -130.1484,B 24.9021,C -2.2848,E1 24.909,E2 -145.5673} C_DIS
LIN {X -40.1878,Y -54.088,Z 76,A -133.3752,B 24.9031,C -2.2726,E1 24.9016,E2 -142.2998} C_DIS
LIN {X -42.7527,Y -52.0847,Z 76,A -135.1716,B 24.9009,C -2.2985,E1 24.8979,E2 -140.5585} C_DIS
LIN {X -45.1789,Y -49.9941,Z 76,A -137.9065,B 24.9005,C -2.3035,E1 24.8921,E2 -137.8247} C_DIS
LIN {X -46.8633,Y -48.418,Z 76,A -140.3557,B 24.901,C -2.297,E1 24.8871,E2 -135.35} C_DIS
LIN {X -48.8188,Y -46.447,Z 76,A -142.8941,B 24.901,C -2.2982,E1 24.8822,E2 -132.8036} C_DIS
LIN {X -51.4469,Y -43.5168,Z 76,A -145.9161,B 24.8997,C -2.3126,E1 24.8767,E2 -129.8022} C_DIS
LIN {X -53.7197,Y -40.678,Z 76,A -148.5965,B 24.8983,C -2.3286,E1 24.8721,E2 -127.1472} C_DIS
LIN {X -55.5252,Y -38.1774,Z 76,A -151.6547,B 24.8985,C -2.3258,E1 24.8671,E2 -124.0676} C_DIS
LIN {X -57.1735,Y -35.66,Z 76,A -154.2458,B 24.898,C -2.3317,E1 24.8632,E2 -121.4774} C_DIS
LIN {X -59.8336,Y -30.9922,Z 76,A -159.3869,B 24.898,C -2.3321,E1 24.8563,E2 -116.3101} C_DIS
LIN {X -61.4698,Y -27.6029,Z 76,A -162.0016,B 24.8961,C -2.353,E1 24.8532,E2 -113.731} C_DIS
LIN {X -62.6498,Y -24.8088,Z 76,A -164.1679,B 24.8947,C -2.3688,E1 24.8509,E2 -111.5904} C_DIS
LIN {X -63.3993,Y -22.8265,Z 76,A -166.4911,B 24.8952,C -2.3633,E1 24.8487,E2 -109.2411} C_DIS
LIN {X -64.42,Y -19.7622,Z 76,A -169.3162,B 24.8946,C -2.3698,E1 24.8463,E2 -106.4152} C_DIS
LIN {X -65.5315,Y -15.689,Z 76,A -172.8421,B 24.8935,C -2.382,E1 24.8438,E2 -102.8978} C_DIS
LIN {X -66.1557,Y -12.8013,Z 76,A -175.3657,B 24.8929,C -2.3894,E1 24.8424,E2 -100.3771} C_DIS
LIN {X -66.8983,Y -8.0693,Z 76,A -179.0611,B 24.891,C -2.4097,E1 24.8409,E2 -96.7081} C_DIS
LIN {X -67.213,Y -4.7862,Z 76,A 177.4505,B 24.8915,C -2.4047,E1 24.84,E2 -93.1868} C_DIS
LIN {X -67.3625,Y -1.6944,Z 76,A 174.9604,B 24.8905,C -2.4158,E1 24.8398,E2 -90.7083} C_DIS
LIN {X -67.3668,Y 1.4894,Z 76,A 172.38,B 24.8895,C -2.4269,E1 24.8398,E2 -88.139} C_DIS
LIN {X -67.169,Y 5.3632,Z 76,A 169.2148,B 24.8883,C -2.4401,E1 24.8404,E2 -84.9861} C_DIS
LIN {X -66.918,Y 7.9012,Z 76,A 166.8507,B 24.888,C -2.443,E1 24.8411,E2 -82.6148} C_DIS
LIN {X -66.108,Y 13.049,Z 76,A 162.5529,B 24.8865,C -2.4596,E1 24.8431,E2 -78.3313} C_DIS
LIN {X -65.1364,Y 17.2567,Z 76,A 159.0046,B 24.8852,C -2.4736,E1 24.8454,E2 -74.7955} C_DIS
LIN {X -64.5194,Y 19.4363,Z 76,A 156.7209,B 24.8852,C -2.4724,E1 24.8471,E2 -72.4956} C_DIS
LIN {X -63.6334,Y 22.1644,Z 76,A 154.3467,B 24.8845,C -2.4812,E1 24.8493,E2 -70.129} C_DIS
LIN {X -61.4293,Y 27.6927,Z 76,A 149.1548,B 24.8833,C -2.4937,E1 24.8548,E2 -64.9381} C_DIS
LIN {X -59.7697,Y 31.1148,Z 76,A 146.0189,B 24.8822,C -2.5051,E1 24.8586,E2 -61.8127} C_DIS
LIN {X -58.4978,Y 33.4436,Z 76,A 143.6813,B 24.8817,C -2.5099,E1 24.8618,E2 -59.4743} C_DIS
LIN {X -57.0181,Y 35.9088,Z 76,A 140.8477,B 24.8818,C -2.5089,E1 24.866,E2 -56.6237} C_DIS
LIN {X -54.3298,Y 39.8587,Z 76,A 137.3187,B 24.8798,C -2.5308,E1 24.8716,E2 -53.1296} C_DIS
LIN {X -53.3576,Y 41.151,Z 76,A 135.6994,B 24.8799,C -2.5294,E1 24.8744,E2 -51.4993} C_DIS
LIN {X -51.4241,Y 43.5437,Z 76,A 132.3166,B 24.8808,C -2.5204,E1 24.8805,E2 -48.0794} C_DIS
LIN {X -49.1544,Y 46.0901,Z 76,A 130.0495,B 24.8788,C -2.5405,E1 24.8847,E2 -45.8503} C_DIS
LIN {X -46.4404,Y 48.825,Z 76,A 126.8441,B 24.878,C -2.5497,E1 24.8911,E2 -42.6534} C_DIS
LIN {X -44.0716,Y 50.9731,Z 76,A 123.4398,B 24.8787,C -2.5415,E1 24.8983,E2 -39.2163} C_DIS
LIN {X -41.5676,Y 53.0344,Z 76,A 121.081,B 24.8774,C -2.5557,E1 24.9034,E2 -36.8825} C_DIS
LIN {X -39.3192,Y 54.722,Z 76,A 118.9671,B 24.8764,C -2.5663,E1 24.9082,E2 -34.7866} C_DIS
LIN {X -36.712,Y 56.5049,Z 76,A 116.3074,B 24.8758,C -2.572,E1 24.9143,E2 -32.1316} C_DIS
LIN {X -34.3008,Y 57.9991,Z 76,A 113.4114,B 24.8764,C -2.5661,E1 24.9213,E2 -29.2126} C_DIS
LIN {X -30.4702,Y 60.1004,Z 76,A 110.1488,B 24.8748,C -2.5819,E1 24.9293,E2 -25.9787} C_DIS
LIN {X -25.6471,Y 62.3116,Z 76,A 105.9953,B 24.8734,C -2.5963,E1 24.9398,E2 -21.8495} C_DIS
LIN {X -23.0155,Y 63.3304,Z 76,A 103.4667,B 24.8734,C -2.5966,E1 24.9464,E2 -19.3163} C_DIS
LIN {X -20.7897,Y 64.0955,Z 76,A 100.6919,B 24.8748,C -2.582,E1 24.9539,E2 -16.5016} C_DIS
LIN {X -15.8048,Y 65.5033,Z 76,A 97.0762,B 24.8727,C -2.6039,E1 24.9635,E2 -12.9325} C_DIS
LIN {X -12.1011,Y 66.2875,Z 76,A 92.9695,B 24.8744,C -2.5867,E1 24.9749,E2 -8.7802} C_DIS
LIN {X -8.4995,Y 66.8448,Z 76,A 90.2221,B 24.8734,C -2.5965,E1 24.9824,E2 -6.054} C_DIS
LIN {X -4.6957,Y 67.2192,Z 76,A 87.3162,B 24.8725,C -2.6058,E1 24.9905,E2 -3.1689} C_DIS
LIN {X -2.1507,Y 67.3484,Z 76,A 84.7938,B 24.8732,C -2.5984,E1 24.9975,E2 -0.6283} C_DIS
LIN {X 2.5049,Y 67.3374,Z 76,A 80.3157,B 24.8744,C -2.587,E1 25.0101,E2 3.8762} C_DIS
LIN {X 5.8247,Y 67.1312,Z 76,A 78.4168,B 24.8723,C -2.6083,E1 25.0153,E2 5.7233} C_DIS
LIN {X 8.7375,Y 66.814,Z 76,A 75.5886,B 24.8731,C -2.6,E1 25.0232,E2 8.5692} C_DIS
LIN {X 11.3318,Y 66.4235,Z 76,A 73.555,B 24.8727,C -2.6039,E1 25.0287,E2 10.5914} C_DIS
LIN {X 16.0299,Y 65.4484,Z 76,A 69.3003,B 24.8733,C -2.5978,E1 25.0404,E2 14.8551} C_DIS
LIN {X 19.6704,Y 64.4485,Z 76,A 66.2013,B 24.8733,C -2.5982,E1 25.0487,E2 17.9478} C_DIS
LIN {X 22.7221,Y 63.4374,Z 76,A 63.1705,B 24.8742,C -2.5888,E1 25.0567,E2 20.995} C_DIS
LIN {X 26.02,Y 62.1565,Z 76,A 60.5564,B 24.8735,C -2.5953,E1 25.0634,E2 23.5876} C_DIS
LIN {X 28.7991,Y 60.9197,Z 76,A 57.6246,B 24.8747,C -2.5839,E1 25.0709,E2 26.5391} C_DIS
LIN {X 33.5674,Y 58.4266,Z 76,A 53.6332,B 24.8738,C -2.5923,E1 25.0806,E2 30.4993} C_DIS
LIN {X 35.5358,Y 57.2511,Z 76,A 51.453,B 24.8747,C -2.5836,E1 25.0859,E2 32.6932} C_DIS
LIN {X 38.8245,Y 55.075,Z 76,A 48.0343,B 24.8754,C -2.5766,E1 25.0938,E2 36.117} C_DIS
LIN {X 41.2351,Y 53.2929,Z 76,A 44.7819,B 24.8775,C -2.5546,E1 25.1011,E2 39.4097} C_DIS
LIN {X 43.8547,Y 51.1591,Z 76,A 43.1926,B 24.8749,C -2.5815,E1 25.1043,E2 40.9292} C_DIS
LIN {X 45.9268,Y 49.308,Z 76,A 40.3383,B 24.8766,C -2.5643,E1 25.1103,E2 43.8128} C_DIS
LIN {X 49.2973,Y 45.9382,Z 76,A 36.6781,B 24.8764,C -2.5657,E1 25.1175,E2 47.4539} C_DIS
LIN {X 51.1946,Y 43.813,Z 76,A 34.034,B 24.8775,C -2.5546,E1 25.1224,E2 50.1124} C_DIS
LIN {X 52.8882,Y 41.7526,Z 76,A 30.9719,B 24.8799,C -2.5289,E1 25.1278,E2 53.221} C_DIS
LIN {X 55.6172,Y 38.0431,Z 76,A 27.7223,B 24.8792,C -2.5364,E1 25.133,E2 56.4371} C_DIS
LIN {X 57.2685,Y 35.5079,Z 76,A 24.4189,B 24.8817,C -2.5109,E1 25.1379,E2 59.7841} C_DIS
LIN {X 58.9755,Y 32.5948,Z 76,A 22.3145,B 24.8805,C -2.5231,E1 25.1408,E2 61.8486} C_DIS
LIN {X 60.2748,Y 30.1237,Z 76,A 19.7883,B 24.8815,C -2.5126,E1 25.144,E2 64.3861} C_DIS
LIN {X 62.2797,Y 25.7255,Z 76,A 15.8594,B 24.8821,C -2.5058,E1 25.1484,E2 68.3098} C_DIS
LIN {X 63.4268,Y 22.7512,Z 76,A 12.4124,B 24.8847,C -2.4786,E1 25.1517,E2 71.8017} C_DIS
LIN {X 64.4925,Y 19.5262,Z 76,A 10.5559,B 24.8829,C -2.4972,E1 25.1532,E2 73.6038} C_DIS
LIN {X 65.5514,Y 15.6067,Z 76,A 7.0228,B 24.8841,C -2.4847,E1 25.1558,E2 77.1462} C_DIS
LIN {X 66.3828,Y 11.5716,Z 76,A 2.8994,B 24.8867,C -2.4575,E1 25.1579,E2 81.3098} C_DIS
LIN {X 67.0095,Y 7.0837,Z 76,A -0.3482,B 24.8863,C -2.4615,E1 25.1591,E2 84.5286} C_DIS
LIN {X 67.2634,Y 4.0206,Z 76,A -3.0222,B 24.8872,C -2.4517,E1 25.1596,E2 87.2099} C_DIS
LIN {X 67.3763,Y 0.972,Z 76,A -5.5769,B 24.8878,C -2.4445,E1 25.1598,E2 89.7663} C_DIS
LIN {X 67.3512,Y -2.0628,Z 76,A -8.7136,B 24.89,C -2.4216,E1 25.1596,E2 92.9388} C_DIS
LIN {X 67.0718,Y -6.4725,Z 76,A -11.9413,B 24.8898,C -2.4237,E1 25.1589,E2 96.1422} C_DIS
LIN {X 66.593,Y -10.2867,Z 76,A -15.4376,B 24.8912,C -2.4073,E1 25.1575,E2 99.6566} C_DIS
LIN {X 65.9143,Y -13.995,Z 76,A -18.4729,B 24.8918,C -2.4017,E1 25.1559,E2 102.6874} C_DIS
LIN {X 65.0559,Y -17.5547,Z 76,A -21.459,B 24.8923,C -2.3954,E1 25.1538,E2 105.6712} C_DIS
LIN {X 63.961,Y -21.2015,Z 76,A -24.5879,B 24.893,C -2.3883,E1 25.1512,E2 108.7992} C_DIS
LIN {X 63.1767,Y -23.4368,Z 76,A -26.5464,B 24.8934,C -2.3836,E1 25.1493,E2 110.7577} C_DIS
LIN {X 62.1956,Y -25.9271,Z 76,A -28.879,B 24.8941,C -2.3752,E1 25.1469,E2 113.0973} C_DIS
LIN {X 60.4212,Y -29.8283,Z 76,A -32.3216,B 24.8946,C -2.3698,E1 25.1428,E2 116.5341} C_DIS
LIN {X 59.5252,Y -31.5791,Z 76,A -34.3096,B 24.8958,C -2.3565,E1 25.1402,E2 118.543} C_DIS
LIN {X 57.5515,Y -35.0467,Z 76,A -37.3786,B 24.8958,C -2.3554,E1 25.1359,E2 121.5987} C_DIS
LIN {X 55.5536,Y -38.1338,Z 76,A -40.8973,B 24.8976,C -2.3364,E1 25.1305,E2 125.1448} C_DIS
LIN {X 53.1445,Y -41.4256,Z 76,A -44.4239,B 24.8985,C -2.3257,E1 25.1245,E2 128.68} C_DIS
LIN {X 51.0406,Y -43.9937,Z 76,A -46.803,B 24.8981,C -2.33,E1 25.1203,E2 131.038} C_DIS
LIN {X 48.8063,Y -46.4584,Z 76,A -49.8772,B 24.8993,C -2.3166,E1 25.1144,E2 134.1304} C_DIS
LIN {X 46.1112,Y -49.1345,Z 76,A -53.224,B 24.9002,C -2.3059,E1 25.1076,E2 137.4885} C_DIS
LIN {X 43.6243,Y -51.3553,Z 76,A -55.5375,B 24.8996,C -2.313,E1 25.1028,E2 139.7761} C_DIS
LIN {X 41.1888,Y -53.3285,Z 76,A -58.6394,B 24.9011,C -2.2961,E1 25.096,E2 142.9066} C_DIS
LIN {X 38.9645,Y -54.975,Z 76,A -61.0609,B 24.9017,C -2.2895,E1 25.0905,E2 145.3351} C_DIS
LIN {X 35.2,Y -57.4583,Z 76,A -64.9587,B 24.9024,C -2.2807,E1 25.0813,E2 149.2413} C_DIS
LIN {X 31.4069,Y -59.6159,Z 76,A -68.4158,B 24.9024,C -2.2807,E1 25.0728,E2 152.6884} C_DIS
LIN {X 28.266,Y -61.1679,Z 76,A -71.2427,B 24.9024,C -2.2798,E1 25.0657,E2 155.5099} C_DIS
LIN {X 23.929,Y -62.9908,Z 76,A -75.1405,B 24.9028,C -2.2767,E1 25.0556,E2 159.406} C_DIS
LIN {X 20.7416,Y -64.1111,Z 76,A -78.12,B 24.9033,C -2.2705,E1 25.0477,E2 162.3944} C_DIS
LIN {X 18.4785,Y -64.7997,Z 76,A -80.2487,B 24.9037,C -2.2654,E1 25.042,E2 164.5317} C_DIS
LIN {X 14.9547,Y -65.7027,Z 76,A -83.2727,B 24.9038,C -2.2641,E1 25.0338,E2 167.5543} C_DIS
LIN {X 11.6811,Y -66.3631,Z 76,A -86.3391,B 24.9045,C -2.2563,E1 25.0253,E2 170.6358} C_DIS
LIN {X 7.1925,Y -66.9981,Z 76,A -89.9201,B 24.9041,C -2.2605,E1 25.0155,E2 174.204} C_DIS
LIN {X 4.0639,Y -67.261,Z 76,A -92.254,B 24.9036,C -2.2673,E1 25.009,E2 176.5205} C_DIS
LIN {X 1.6849,Y -67.3628,Z 76,A -94.5836,B 24.9042,C -2.2593,E1 25.0025,E2 178.8685} C_DIS
LIN {X 1.6849,Y -67.3628,Z 76,A -94.5836,B 24.9042,C -2.2593,E1 25.0025,E2 178.8685} C_DIS
Enddeposition()
LIN {X 0.4208,Y -66.4032,Z 76,A -94.9923,B 24.9014,C -2.292,E1 25.0015,E2 179.1997} C_DIS
Startdeposition()
$VEL.CP = VEL_PRINT
LIN {X 2.5655,Y -66.3589,Z 76,A -92.6689,B 24.9004,C -2.3038,E1 25.0081,E2 176.8486} C_DIS
LIN {X 5.1298,Y -66.2095,Z 76,A -90.4912,B 24.9004,C -2.3038,E1 25.0142,E2 174.6717} C_DIS
LIN {X 9.1851,Y -65.7698,Z 76,A -86.3603,B 24.8989,C -2.321,E1 25.0257,E2 170.5035} C_DIS
LIN {X 12.5519,Y -65.2109,Z 76,A -83.4277,B 24.8987,C -2.3231,E1 25.0338,E2 167.5693} C_DIS
LIN {X 18.2797,Y -63.8427,Z 76,A -78.5059,B 24.8987,C -2.3242,E1 25.0471,E2 162.6523} C_DIS
LIN {X 22.3787,Y -62.5249,Z 76,A -75.1781,B 24.8991,C -2.3191,E1 25.0558,E2 159.3432} C_DIS
LIN {X 25.0355,Y -61.508,Z 76,A -72.5854,B 24.8985,C -2.326,E1 25.0626,E2 156.74} C_DIS
LIN {X 28.1441,Y -60.1493,Z 76,A -69.8402,B 24.8985,C -2.3258,E1 25.0695,E2 154.0021} C_DIS
LIN {X 30.7469,Y -58.8616,Z 76,A -67.5669,B 24.8987,C -2.324,E1 25.0752,E2 151.7392} C_DIS
LIN {X 33.4168,Y -57.3888,Z 76,A -64.6206,B 24.8976,C -2.3367,E1 25.0824,E2 148.7716} C_DIS
LIN {X 36.1608,Y -55.7003,Z 76,A -61.8651,B 24.8971,C -2.3413,E1 25.0889,E2 146.0141} C_DIS
LIN {X 38.8973,Y -53.8253,Z 76,A -58.7072,B 24.896,C -2.3547,E1 25.0961,E2 142.8354} C_DIS
LIN {X 42.6254,Y -50.9229,Z 76,A -55.2779,B 24.8967,C -2.3467,E1 25.1036,E2 139.4378} C_DIS
LIN {X 45.2184,Y -48.6335,Z 76,A -51.7785,B 24.8949,C -2.367,E1 25.1109,E2 135.9045} C_DIS
LIN {X 48.2823,Y -45.593,Z 76,A -47.8612,B 24.8936,C -2.3811,E1 25.1185,E2 131.9706} C_DIS
LIN {X 50.5861,Y -43.0239,Z 76,A -45.0683,B 24.8934,C -2.3838,E1 25.1236,E2 129.1841} C_DIS
LIN {X 53.2911,Y -39.6254,Z 76,A -41.9188,B 24.8939,C -2.3779,E1 25.129,E2 126.0634} C_DIS
LIN {X 55.9196,Y -35.8192,Z 76,A -37.6593,B 24.8923,C -2.3959,E1 25.1357,E2 121.7822} C_DIS
LIN {X 57.455,Y -33.3016,Z 76,A -35.1629,B 24.8917,C -2.4019,E1 25.1392,E2 119.2846} C_DIS
LIN {X 58.5138,Y -31.4043,Z 76,A -32.5833,B 24.8895,C -2.4262,E1 25.1427,E2 116.6611} C_DIS
LIN {X 60.6382,Y -27.0752,Z 76,A -29.2578,B 24.8904,C -2.4161,E1 25.1466,E2 113.3775} C_DIS
LIN {X 61.6572,Y -24.6687,Z 76,A -26.8702,B 24.8895,C -2.4264,E1 25.1491,E2 110.9785} C_DIS
LIN {X 62.8268,Y -21.5152,Z 76,A -23.5011,B 24.8875,C -2.4479,E1 25.1523,E2 107.5776} C_DIS
LIN {X 64.4374,Y -16.0604,Z 76,A -18.6039,B 24.8862,C -2.4629,E1 25.1559,E2 102.6731} C_DIS
LIN {X 65.1756,Y -12.7353,Z 76,A -15.7249,B 24.8854,C -2.4705,E1 25.1574,E2 99.7929} C_DIS
LIN {X 66.0004,Y -7.3546,Z 76,A -11.593,B 24.8854,C -2.4701,E1 25.159,E2 95.6863} C_DIS
LIN {X 66.304,Y -3.7135,Z 76,A -8.1284,B 24.8838,C -2.4886,E1 25.1597,E2 92.1986} C_DIS
LIN {X 66.4083,Y 0.1704,Z 76,A -5.0748,B 24.8835,C -2.4911,E1 25.1597,E2 89.1572} C_DIS
LIN {X 66.3344,Y 3.1371,Z 76,A -2.4853,B 24.8827,C -2.5,E1 25.1595,E2 86.5621} C_DIS
LIN {X 66.0879,Y 6.523,Z 76,A 0.3579,B 24.882,C -2.5069,E1 25.1588,E2 83.7195} C_DIS
LIN {X 65.838,Y 8.683,Z 76,A 2.8841,B 24.8798,C -2.5303,E1 25.1579,E2 81.153} C_DIS
LIN {X 65.058,Y 13.3217,Z 76,A 6.216,B 24.8805,C -2.5232,E1 25.1562,E2 77.8573} C_DIS
LIN {X 64.3903,Y 16.2475,Z 76,A 8.5578,B 24.8804,C -2.5245,E1 25.1547,E2 75.526} C_DIS
LIN {X 63.2689,Y 20.1776,Z 76,A 12.5102,B 24.8783,C -2.5463,E1 25.1515,E2 71.5446} C_DIS
LIN {X 62.1434,Y 23.414,Z 76,A 15.1739,B 24.8783,C -2.5471,E1 25.149,E2 68.8938} C_DIS
LIN {X 61.1203,Y 25.9684,Z 76,A 17.4096,B 24.8779,C -2.5502,E1 25.1466,E2 66.6631} C_DIS
LIN {X 60.0516,Y 28.354,Z 76,A 19.89,B 24.8767,C -2.5624,E1 25.1437,E2 64.1673} C_DIS
LIN {X 58.7898,Y 30.8832,Z 76,A 22.2377,B 24.8763,C -2.5667,E1 25.1407,E2 61.822} C_DIS
LIN {X 56.9469,Y 34.1641,Z 76,A 25.5387,B 24.8754,C -2.5767,E1 25.1361,E2 58.5145} C_DIS
LIN {X 55.2988,Y 36.7711,Z 76,A 28.153,B 24.8748,C -2.5822,E1 25.1321,E2 55.9} C_DIS
LIN {X 53.5915,Y 39.2168,Z 76,A 30.5853,B 24.8746,C -2.5849,E1 25.1282,E2 53.4732} C_DIS
LIN {X 51.812,Y 41.5409,Z 76,A 33.2345,B 24.8737,C -2.5941,E1 25.1236,E2 50.8148} C_DIS
LIN {X 50.3714,Y 43.2759,Z 76,A 35.2167,B 24.8731,C -2.5995,E1 25.12,E2 48.8289} C_DIS
LIN {X 48.2847,Y 45.5918,Z 76,A 37.6108,B 24.8733,C -2.5978,E1 25.1155,E2 46.4493} C_DIS
LIN {X 46.2747,Y 47.6312,Z 76,A 40.3177,B 24.8722,C -2.609,E1 25.1101,E2 43.7274} C_DIS
LIN {X 43.8185,Y 49.8997,Z 76,A 43.1397,B 24.8718,C -2.6131,E1 25.1043,E2 40.9069} C_DIS
LIN {X 41.9482,Y 51.4819,Z 76,A 45.4801,B 24.8708,C -2.6228,E1 25.0992,E2 38.5526} C_DIS
LIN {X 39.2259,Y 53.5849,Z 76,A 48.0528,B 24.8713,C -2.618,E1 25.0935,E2 36.0005} C_DIS
LIN {X 36.8297,Y 55.2602,Z 76,A 50.7354,B 24.8705,C -2.6261,E1 25.0873,E2 33.3078} C_DIS
LIN {X 34.3621,Y 56.8267,Z 76,A 53.2599,B 24.8701,C -2.6299,E1 25.0813,E2 30.7822} C_DIS
LIN {X 31.9287,Y 58.2293,Z 76,A 55.7056,B 24.8697,C -2.6338,E1 25.0753,E2 28.3346} C_DIS
LIN {X 28.5359,Y 59.9648,Z 76,A 59.0102,B 24.8693,C -2.6382,E1 25.0671,E2 25.0283} C_DIS
LIN {X 25.6872,Y 61.2388,Z 76,A 61.3929,B 24.8698,C -2.6336,E1 25.061,E2 22.6624} C_DIS
LIN {X 23.2111,Y 62.2203,Z 76,A 63.9346,B 24.869,C -2.6417,E1 25.0544,E2 20.107} C_DIS
LIN {X 20.3668,Y 63.2077,Z 76,A 66.5013,B 24.8688,C -2.6431,E1 25.0476,E2 17.5419} C_DIS
LIN {X 17.5272,Y 64.0535,Z 76,A 69.0763,B 24.8686,C -2.6453,E1 25.0407,E2 14.9661} C_DIS
LIN {X 14.8062,Y 64.7364,Z 76,A 71.6114,B 24.8682,C -2.6493,E1 25.0337,E2 12.425} C_DIS
LIN {X 11.5474,Y 65.3966,Z 76,A 74.3447,B 24.8684,C -2.6472,E1 25.0263,E2 9.6997} C_DIS
LIN {X 8.9892,Y 65.7976,Z 76,A 76.9749,B 24.8674,C -2.6572,E1 25.0189,E2 7.0482} C_DIS
LIN {X 4.3214,Y 66.2673,Z 76,A 81.1588,B 24.8671,C -2.6606,E1 25.0073,E2 2.8583} C_DIS
LIN {X -0.1772,Y 66.4081,Z 76,A 84.2999,B 24.8689,C -2.6428,E1 24.9986,E2 -0.2399} C_DIS
LIN {X -2.8594,Y 66.3463,Z 76,A 86.9076,B 24.8683,C -2.6488,E1 24.9913,E2 -2.8625} C_DIS
LIN {X -6.5934,Y 66.0805,Z 76,A 90.0705,B 24.8686,C -2.6458,E1 24.9825,E2 -6.0196} C_DIS
LIN {X -9.6571,Y 65.7027,Z 76,A 92.7479,B 24.8686,C -2.6445,E1 24.9751,E2 -8.6959} C_DIS
LIN {X -15.2541,Y 64.633,Z 76,A 97.6737,B 24.8691,C -2.6406,E1 24.9617,E2 -13.6182} C_DIS
LIN {X -19.9966,Y 63.3266,Z 76,A 101.9733,B 24.8694,C -2.6373,E1 24.9501,E2 -17.9169} C_DIS
LIN {X -23.1433,Y 62.2458,Z 76,A 104.8392,B 24.8698,C -2.6336,E1 24.9426,E2 -20.7797} C_DIS
LIN {X -25.5774,Y 61.2851,Z 76,A 107.9696,B 24.8682,C -2.6498,E1 24.9344,E2 -23.9557} C_DIS
LIN {X -28.949,Y 59.7663,Z 76,A 110.2352,B 24.8707,C -2.6246,E1 24.9288,E2 -26.167} C_DIS
LIN {X -31.438,Y 58.4955,Z 76,A 112.7007,B 24.8709,C -2.6218,E1 24.9227,E2 -28.6326} C_DIS
LIN {X -34.0814,Y 56.9963,Z 76,A 115.344,B 24.8714,C -2.6176,E1 24.9164,E2 -31.2739} C_DIS
LIN {X -36.4977,Y 55.4791,Z 76,A 117.7919,B 24.8718,C -2.6127,E1 24.9106,E2 -33.7181} C_DIS
LIN {X -38.9717,Y 53.7709,Z 76,A 120.4274,B 24.8723,C -2.6084,E1 24.9046,E2 -36.3524} C_DIS
LIN {X -41.4478,Y 51.8861,Z 76,A 123.2365,B 24.8725,C -2.6054,E1 24.8984,E2 -39.1647} C_DIS
LIN {X -44.0193,Y 49.7237,Z 76,A 126.0184,B 24.8734,C -2.5965,E1 24.8926,E2 -41.9362} C_DIS
LIN {X -46.2053,Y 47.6981,Z 76,A 128.6116,B 24.874,C -2.591,E1 24.8873,E2 -44.527} C_DIS
LIN {X -47.7802,Y 46.1201,Z 76,A 130.6866,B 24.8741,C -2.5896,E1 24.8833,E2 -46.6074} C_DIS
LIN {X -50.3578,Y 43.2919,Z 76,A 133.8159,B 24.8753,C -2.5777,E1 24.8775,E2 -49.7224} C_DIS
LIN {X -52.2327,Y 41.0097,Z 76,A 136.4244,B 24.8758,C -2.5724,E1 24.873,E2 -52.3303} C_DIS
LIN {X -54.0716,Y 38.5522,Z 76,A 139.335,B 24.8759,C -2.5707,E1 24.8682,E2 -55.2511} C_DIS
LIN {X -56.1063,Y 35.5282,Z 76,A 142.2856,B 24.8772,C -2.558,E1 24.8637,E2 -58.1863} C_DIS
LIN {X -57.5912,Y 33.0646,Z 76,A 144.6252,B 24.8781,C -2.5481,E1 24.8604,E2 -60.5143} C_DIS
LIN {X -58.9524,Y 30.574,Z 76,A 147.1831,B 24.8786,C -2.5433,E1 24.857,E2 -63.0741} C_DIS
LIN {X -60.0559,Y 28.3448,Z 76,A 149.1822,B 24.8795,C -2.534,E1 24.8546,E2 -65.0619} C_DIS
LIN {X -61.4804,Y 25.1032,Z 76,A 152.4128,B 24.88,C -2.5284,E1 24.8511,E2 -68.2971} C_DIS
LIN {X -62.5105,Y 22.4183,Z 76,A 154.9737,B 24.8806,C -2.5225,E1 24.8486,E2 -70.8582} C_DIS
LIN {X -63.4917,Y 19.4641,Z 76,A 157.6511,B 24.8814,C -2.5141,E1 24.8463,E2 -73.5309} C_DIS
LIN {X -64.3175,Y 16.531,Z 76,A 159.8106,B 24.883,C -2.4965,E1 24.8447,E2 -75.6609} C_DIS
LIN {X -64.8707,Y 14.2056,Z 76,A 162.3528,B 24.8827,C -2.4996,E1 24.8431,E2 -78.2256} C_DIS
LIN {X -65.5763,Y 10.4821,Z 76,A 165.6454,B 24.8836,C -2.4898,E1 24.8415,E2 -81.5142} C_DIS
LIN {X -65.9582,Y 7.7151,Z 76,A 168.0664,B 24.8843,C -2.4824,E1 24.8407,E2 -83.932} C_DIS
LIN {X -66.2321,Y 4.8419,Z 76,A 170.5541,B 24.8851,C -2.4744,E1 24.8401,E2 -86.4156} C_DIS
LIN {X -66.3705,Y 2.2387,Z 76,A 173.3096,B 24.8848,C -2.4776,E1 24.8398,E2 -89.1953} C_DIS
LIN {X -66.3802,Y -1.9219,Z 76,A 176.4698,B 24.8866,C -2.4575,E1 24.8399,E2 -92.3265} C_DIS
LIN {X -66.0268,Y -7.1069,Z 76,A -179.0971,B 24.888,C -2.4424,E1 24.8409,E2 -96.7501} C_DIS
LIN {X -65.5825,Y -10.442,Z 76,A -176.0288,B 24.8886,C -2.4367,E1 24.8421,E2 -99.8231} C_DIS
LIN {X -65.0154,Y -13.529,Z 76,A -173.3356,B 24.8894,C -2.4281,E1 24.8436,E2 -102.5117} C_DIS
LIN {X -64.3109,Y -16.5565,Z 76,A -170.6825,B 24.8901,C -2.4195,E1 24.8453,E2 -105.1597} C_DIS
LIN {X -63.5518,Y -19.2701,Z 76,A -168.0974,B 24.8905,C -2.4153,E1 24.8474,E2 -107.7499} C_DIS
LIN {X -62.4992,Y -22.449,Z 76,A -165.3404,B 24.8915,C -2.4042,E1 24.8498,E2 -110.4959} C_DIS
LIN {X -61.5113,Y -25.0273,Z 76,A -162.8417,B 24.8919,C -2.3998,E1 24.8524,E2 -112.9981} C_DIS
LIN {X -60.2962,Y -27.8284,Z 76,A -160.1875,B 24.8926,C -2.3928,E1 24.8555,E2 -115.6501} C_DIS
LIN {X -58.8962,Y -30.6812,Z 76,A -157.5942,B 24.8935,C -2.3823,E1 24.8587,E2 -118.2322} C_DIS
LIN {X -57.2534,Y -33.6464,Z 76,A -154.6453,B 24.8942,C -2.375,E1 24.8628,E2 -121.1792} C_DIS
LIN {X -55.8762,Y -35.8868,Z 76,A -152.2274,B 24.8944,C -2.3723,E1 24.8664,E2 -123.603} C_DIS
LIN {X -54.2134,Y -38.3535,Z 76,A -149.5283,B 24.8947,C -2.3688,E1 24.8707,E2 -126.3069} C_DIS
LIN {X -52.1434,Y -41.1227,Z 76,A -146.7293,B 24.8957,C -2.3578,E1 24.8754,E2 -129.0929} C_DIS
LIN {X -50.2604,Y -43.4054,Z 76,A -144.0768,B 24.896,C -2.3541,E1 24.8802,E2 -131.7487} C_DIS
LIN {X -47.9637,Y -45.9297,Z 76,A -141.1743,B 24.8967,C -2.3468,E1 24.8857,E2 -134.6467} C_DIS
LIN {X -45.8807,Y -48.0109,Z 76,A -138.5898,B 24.897,C -2.3425,E1 24.8909,E2 -137.2317} C_DIS
LIN {X -43.7571,Y -49.9533,Z 76,A -136.0482,B 24.8973,C -2.339,E1 24.8962,E2 -139.775} C_DIS
LIN {X -41.9767,Y -51.4588,Z 76,A -133.9361,B 24.8975,C -2.3375,E1 24.9007,E2 -141.8915} C_DIS
LIN {X -39.2676,Y -53.5543,Z 76,A -131.1246,B 24.8982,C -2.3292,E1 24.907,E2 -144.6935} C_DIS
LIN {X -36.7875,Y -55.288,Z 76,A -128.5617,B 24.8987,C -2.324,E1 24.9129,E2 -147.2526} C_DIS
LIN {X -34.6979,Y -56.6227,Z 76,A -126.3589,B 24.8988,C -2.3222,E1 24.9181,E2 -149.458} C_DIS
LIN {X -30.5093,Y -58.9855,Z 76,A -122.2023,B 24.8993,C -2.3169,E1 24.9283,E2 -153.6138} C_DIS
LIN {X -27.677,Y -60.3667,Z 76,A -119.3694,B 24.8993,C -2.3163,E1 24.9355,E2 -156.4525} C_DIS
LIN {X -24.7555,Y -61.6219,Z 76,A -116.7071,B 24.8997,C -2.3117,E1 24.9423,E2 -159.1099} C_DIS
LIN {X -21.9199,Y -62.686,Z 76,A -114.1256,B 24.9,C -2.3087,E1 24.9491,E2 -161.6895} C_DIS
LIN {X -19.1231,Y -63.5954,Z 76,A -111.6557,B 24.9003,C -2.3053,E1 24.9557,E2 -164.1557} C_DIS
LIN {X -15.9634,Y -64.4611,Z 76,A -108.7431,B 24.9003,C -2.3057,E1 24.9635,E2 -167.0734} C_DIS
LIN {X -13.0915,Y -65.1053,Z 76,A -106.3047,B 24.9006,C -2.3022,E1 24.9702,E2 -169.5065} C_DIS
LIN {X -9.7415,Y -65.6907,Z 76,A -103.0344,B 24.8999,C -2.3092,E1 24.9792,E2 -172.7966} C_DIS
LIN {X -5.6986,Y -66.1642,Z 76,A -99.8551,B 24.9007,C -2.301,E1 24.988,E2 -175.9582} C_DIS
LIN {X -2.9803,Y -66.3411,Z 76,A -97.4638,B 24.9006,C -2.3021,E1 24.9947,E2 -178.3528} C_DIS
LIN {X -0.2014,Y -66.4079,Z 76,A -95.02,B 24.9004,C -2.3037,E1 25.0015,E2 -180.8003} C_DIS
LIN {X -0.2014,Y -66.4079,Z 76,A -95.02,B 24.9004,C -2.3037,E1 25.0015,E2 -180.8003} C_DIS
Enddeposition()
LIN {X 0.4089,Y -65.4292,Z 76,A -94.7808,B 24.8996,C -2.3138,E1 25.0023,E2 -181.0636} C_DIS
Startdeposition()
$VEL.CP = VEL_PRINT
LIN {X -1.6054,Y -65.4145,Z 76,A -97.5347,B 24.9016,C -2.2904,E1 24.9944,E2 -178.2541} C_DIS
LIN {X -4.8218,Y -65.2562,Z 76,A -100.2726,B 24.9014,C -2.2922,E1 24.9868,E2 -175.5195} C_DIS
LIN {X -7.7343,Y -64.9744,Z 76,A -102.8982,B 24.9015,C -2.291,E1 24.9795,E2 -172.8896} C_DIS
LIN {X -10.4188,Y -64.5993,Z 76,A -105.2876,B 24.9015,C -2.2913,E1 24.9729,E2 -170.4986} C_DIS
LIN {X -13.5597,Y -64.0138,Z 76,A -107.9989,B 24.9012,C -2.2943,E1 24.9655,E2 -167.7915} C_DIS
LIN {X -16.225,Y -63.3895,Z 76,A -110.3148,B 24.901,C -2.2974,E1 24.9592,E2 -165.4798} C_DIS
LIN {X -19.0075,Y -62.6126,Z 76,A -113.0244,B 24.9012,C -2.2951,E1 24.9519,E2 -162.7602} C_DIS
LIN {X -22.0485,Y -61.6076,Z 76,A -115.8343,B 24.901,C -2.2972,E1 24.9445,E2 -159.95} C_DIS
LIN {X -25.0372,Y -60.4547,Z 76,A -118.6507,B 24.9008,C -2.2997,E1 24.9372,E2 -157.1333} C_DIS
LIN {X -27.982,Y -59.1493,Z 76,A -121.4746,B 24.9005,C -2.3027,E1 24.93,E2 -154.3097} C_DIS
LIN {X -30.8823,Y -57.6878,Z 76,A -124.3111,B 24.9002,C -2.3065,E1 24.923,E2 -151.4744} C_DIS
LIN {X -33.6478,Y -56.12,Z 76,A -127.1185,B 24.8999,C -2.3099,E1 24.9162,E2 -148.6667} C_DIS
LIN {X -36.3544,Y -54.4058,Z 76,A -129.9351,B 24.8995,C -2.3139,E1 24.9096,E2 -145.8506} C_DIS
LIN {X -38.974,Y -52.561,Z 76,A -132.7519,B 24.8992,C -2.3184,E1 24.9033,E2 -143.0346} C_DIS
LIN {X -41.333,Y -50.7256,Z 76,A -135.3214,B 24.8987,C -2.3241,E1 24.8977,E2 -140.4692} C_DIS
LIN {X -43.6474,Y -48.7481,Z 76,A -138.0565,B 24.8983,C -2.3278,E1 24.8919,E2 -137.7321} C_DIS
LIN {X -45.9808,Y -46.5536,Z 76,A -140.878,B 24.8979,C -2.3331,E1 24.8862,E2 -134.9116} C_DIS
LIN {X -48.2162,Y -44.2343,Z 76,A -143.7093,B 24.8973,C -2.339,E1 24.8808,E2 -132.082} C_DIS
LIN {X -50.3236,Y -41.8212,Z 76,A -146.449,B 24.8967,C -2.3467,E1 24.8759,E2 -129.3481} C_DIS
LIN {X -52.1086,Y -39.5762,Z 76,A -149.0258,B 24.8963,C -2.3513,E1 24.8714,E2 -126.7701} C_DIS
LIN {X -53.9604,Y -37.0123,Z 76,A -151.839,B 24.8957,C -2.3572,E1 24.8669,E2 -123.9572} C_DIS
LIN {X -55.7081,Y -34.3255,Z 76,A -154.6633,B 24.8951,C -2.364,E1 24.8627,E2 -121.1349} C_DIS
LIN {X -57.3295,Y -31.543,Z 76,A -157.4958,B 24.8945,C -2.3712,E1 24.8588,E2 -118.3047} C_DIS
LIN {X -58.8005,Y -28.7076,Z 76,A -160.3172,B 24.8939,C -2.3784,E1 24.8553,E2 -115.4853} C_DIS
LIN {X -60.1399,Y -25.7842,Z 76,A -163.1545,B 24.8932,C -2.3859,E1 24.852,E2 -112.6502} C_DIS
LIN {X -61.3352,Y -22.7952,Z 76,A -165.9853,B 24.8925,C -2.3937,E1 24.8492,E2 -109.8223} C_DIS
LIN {X -62.3781,Y -19.7637,Z 76,A -168.8125,B 24.8918,C -2.4016,E1 24.8467,E2 -106.9977} C_DIS
LIN {X -63.2758,Y -16.6672,Z 76,A -171.6532,B 24.891,C -2.4097,E1 24.8446,E2 -104.1599} C_DIS
LIN {X -64.0159,Y -13.5499,Z 76,A -174.4791,B 24.8903,C -2.4178,E1 24.8429,E2 -101.3368} C_DIS
LIN {X -64.6024,Y -10.3999,Z 76,A -177.3111,B 24.8896,C -2.4259,E1 24.8415,E2 -98.5074} C_DIS
LIN {X -64.9821,Y -7.6687,Z 76,A -179.564,B 24.8886,C -2.4366,E1 24.8407,E2 -96.2666} C_DIS
LIN {X -65.2582,Y -4.794,Z 76,A 177.721,B 24.8882,C -2.4409,E1 24.8401,E2 -93.5456} C_DIS
LIN {X -65.4145,Y -1.6051,Z 76,A 174.9318,B 24.8874,C -2.4498,E1 24.8398,E2 -90.7609} C_DIS
LIN {X -65.4233,Y 1.1291,Z 76,A 172.6632,B 24.8864,C -2.4599,E1 24.8398,E2 -88.5025} C_DIS
LIN {X -65.3103,Y 4.0234,Z 76,A 169.936,B 24.886,C -2.4642,E1 24.8402,E2 -85.7693} C_DIS
LIN {X -65.0354,Y 7.213,Z 76,A 167.1102,B 24.8852,C -2.4726,E1 24.841,E2 -82.9468} C_DIS
LIN {X -64.6047,Y 10.3855,Z 76,A 164.3798,B 24.8843,C -2.4829,E1 24.8421,E2 -80.2246} C_DIS
LIN {X -64.1766,Y 12.7668,Z 76,A 162.2887,B 24.8836,C -2.4901,E1 24.8432,E2 -78.1383} C_DIS
LIN {X -63.6612,Y 15.1286,Z 76,A 160.0221,B 24.8833,C -2.4938,E1 24.8446,E2 -75.8673} C_DIS
LIN {X -62.8446,Y 18.226,Z 76,A 157.1961,B 24.8825,C -2.5021,E1 24.8467,E2 -73.0447} C_DIS
LIN {X -61.8772,Y 21.2799,Z 76,A 154.3708,B 24.8817,C -2.5103,E1 24.8492,E2 -70.2229} C_DIS
LIN {X -60.7618,Y 24.2821,Z 76,A 151.547,B 24.8809,C -2.5184,E1 24.852,E2 -67.4026} C_DIS
LIN {X -59.4915,Y 27.2469,Z 76,A 148.6946,B 24.8802,C -2.5263,E1 24.8552,E2 -64.5533} C_DIS
LIN {X -58.0778,Y 30.143,Z 76,A 145.8636,B 24.8794,C -2.5343,E1 24.8588,E2 -61.7263} C_DIS
LIN {X -56.5323,Y 32.9505,Z 76,A 143.0383,B 24.8787,C -2.542,E1 24.8626,E2 -58.9045} C_DIS
LIN {X -55.0997,Y 35.2917,Z 76,A 140.7956,B 24.8778,C -2.5518,E1 24.8659,E2 -56.6739} C_DIS
LIN {X -53.4883,Y 37.6912,Z 76,A 138.0747,B 24.8775,C -2.555,E1 24.8703,E2 -53.947} C_DIS
LIN {X -51.5811,Y 40.2619,Z 76,A 135.2546,B 24.8768,C -2.562,E1 24.875,E2 -51.1303} C_DIS
LIN {X -49.6989,Y 42.562,Z 76,A 132.6857,B 24.8761,C -2.5693,E1 24.8796,E2 -48.567} C_DIS
LIN {X -47.6527,Y 44.8408,Z 76,A 129.939,B 24.8756,C -2.5746,E1 24.8848,E2 -45.821} C_DIS
LIN {X -45.4029,Y 47.1174,Z 76,A 127.1207,B 24.8749,C -2.581,E1 24.8904,E2 -43.0058} C_DIS
LIN {X -43.0434,Y 49.2823,Z 76,A 124.3825,B 24.8742,C -2.5886,E1 24.8961,E2 -40.275} C_DIS
LIN {X -40.8745,Y 51.0969,Z 76,A 121.8143,B 24.8739,C -2.5921,E1 24.9016,E2 -37.7052} C_DIS
LIN {X -38.3248,Y 53.0362,Z 76,A 118.9958,B 24.8733,C -2.5975,E1 24.9079,E2 -34.8898} C_DIS
LIN {X -35.6827,Y 54.8487,Z 76,A 116.1764,B 24.8728,C -2.6026,E1 24.9145,E2 -32.0732} C_DIS
LIN {X -32.9551,Y 56.5296,Z 76,A 113.3592,B 24.8724,C -2.6074,E1 24.9212,E2 -29.2588} C_DIS
LIN {X -30.4328,Y 57.9251,Z 76,A 110.8751,B 24.8719,C -2.6125,E1 24.9273,E2 -26.7798} C_DIS
LIN {X -27.944,Y 59.1671,Z 76,A 108.386,B 24.8716,C -2.6151,E1 24.9336,E2 -24.2906} C_DIS
LIN {X -25.022,Y 60.4609,Z 76,A 105.5769,B 24.8712,C -2.6189,E1 24.9408,E2 -21.4839} C_DIS
LIN {X -22.0377,Y 61.6114,Z 76,A 102.7676,B 24.8709,C -2.6223,E1 24.9481,E2 -18.677} C_DIS
LIN {X -18.9997,Y 62.615,Z 76,A 99.9435,B 24.8706,C -2.625,E1 24.9556,E2 -15.8543} C_DIS
LIN {X -15.8924,Y 63.4749,Z 76,A 97.1036,B 24.8704,C -2.6275,E1 24.9633,E2 -13.016} C_DIS
LIN {X -12.7381,Y 64.1822,Z 76,A 94.296,B 24.8701,C -2.6304,E1 24.9709,E2 -10.2118} C_DIS
LIN {X -9.5955,Y 64.7268,Z 76,A 91.4959,B 24.8699,C -2.6321,E1 24.9787,E2 -7.4135} C_DIS
LIN {X -6.4286,Y 65.1176,Z 76,A 88.696,B 24.8698,C -2.6335,E1 24.9864,E2 -4.6151} C_DIS
LIN {X -3.2509,Y 65.3532,Z 76,A 85.9048,B 24.8697,C -2.6346,E1 24.9942,E2 -1.8255} C_DIS
LIN {X -0.0839,Y 65.4337,Z 76,A 83.1481,B 24.8696,C -2.6356,E1 25.0019,E2 0.9287} C_DIS
LIN {X 2.9129,Y 65.3682,Z 76,A 80.5072,B 24.8696,C -2.6356,E1 25.0093,E2 3.5694} C_DIS
LIN {X 5.9601,Y 65.161,Z 76,A 78.0063,B 24.8692,C -2.6393,E1 25.0162,E2 6.06} C_DIS
LIN {X 8.8203,Y 64.8369,Z 76,A 75.3099,B 24.8696,C -2.6348,E1 25.0237,E2 8.765} C_DIS
LIN {X 11.9779,Y 64.3286,Z 76,A 72.5991,B 24.8696,C -2.6359,E1 25.0311,E2 11.4703} C_DIS
LIN {X 14.3548,Y 63.8401,Z 76,A 70.3869,B 24.8698,C -2.6329,E1 25.0372,E2 13.6868} C_DIS
LIN {X 17.4616,Y 63.0612,Z 76,A 67.5863,B 24.87,C -2.6312,E1 25.0447,E2 16.487} C_DIS
LIN {X 20.5266,Y 62.1312,Z 76,A 64.7849,B 24.8702,C -2.6291,E1 25.0522,E2 19.2882} C_DIS
Enddeposition()
END
